C03642=1083.822,-32.819,444.005,174.181,18.899,153.143
C03643=1083.816,-33.092,444.020,174.180,18.898,153.143
C03644=1083.809,-33.364,444.033,174.179,18.896,153.143
C03645=1083.803,-33.637,444.048,174.176,18.894,153.143
C03646=1083.796,-33.887,444.060,174.175,18.892,153.143
C03647=1083.791,-34.136,444.072,174.174,18.890,153.143
C03648=1083.785,-34.386,444.084,174.172,18.888,153.143
C03649=1083.779,-34.636,444.097,174.171,18.886,153.143
C03650=1083.773,-34.885,444.109,174.170,18.885,153.143
C03651=1083.767,-35.135,444.122,174.168,18.882,153.143
C03652=1083.762,-35.384,444.134,174.166,18.881,153.143
C03653=1083.756,-35.634,444.147,174.165,18.879,153.143
C03654=1083.750,-35.884,444.159,174.163,18.877,153.142
C03655=1083.743,-36.133,444.172,174.162,18.876,153.142
C03656=1083.738,-36.382,444.184,174.161,18.874,153.142
C03657=1083.732,-36.632,444.197,174.159,18.872,153.142
C03658=1083.726,-36.882,444.209,174.157,18.870,153.142
C03659=1083.721,-37.131,444.221,174.156,18.868,153.142
C03660=1083.715,-37.381,444.234,174.154,18.866,153.142
C03661=1083.708,-37.631,444.246,174.153,18.865,153.142
C03662=1083.702,-37.881,444.259,174.152,18.863,153.142
C03663=1083.697,-38.130,444.271,174.150,18.861,153.142
C03664=1083.691,-38.380,444.283,174.149,18.859,153.142
C03665=1083.685,-38.630,444.296,174.147,18.857,153.142
C03666=1083.680,-38.879,444.308,174.145,18.856,153.142
C03667=1083.673,-39.128,444.320,174.144,18.854,153.141
C03668=1083.668,-39.378,444.333,174.143,18.852,153.141
C03669=1083.662,-39.628,444.345,174.141,18.851,153.141
C03670=1083.656,-39.877,444.357,174.140,18.849,153.141
C03671=1083.650,-40.127,444.369,174.139,18.847,153.141
C03672=1083.644,-40.377,444.381,174.137,18.845,153.141
C03673=1083.637,-40.627,444.393,174.135,18.844,153.141
C03674=1083.632,-40.876,444.405,174.134,18.842,153.141
C03675=1083.626,-41.126,444.418,174.132,18.840,153.141
C03676=1083.620,-41.376,444.430,174.131,18.838,153.141
C03677=1083.614,-41.625,444.442,174.130,18.837,153.141
C03678=1083.608,-41.875,444.454,174.128,18.835,153.141
C03679=1083.602,-42.124,444.466,174.127,18.833,153.141
C03680=1083.596,-42.374,444.479,174.125,18.831,153.141
C03681=1083.590,-42.623,444.491,174.123,18.830,153.141
C03682=1083.584,-42.874,444.502,174.122,18.828,153.140
C03683=1083.578,-43.123,444.515,174.121,18.826,153.140
C03684=1083.572,-43.372,444.527,174.119,18.825,153.140
C03685=1083.566,-43.622,444.539,174.118,18.823,153.140
C03686=1083.560,-43.872,444.552,174.117,18.821,153.140
C03687=1083.554,-44.121,444.563,174.115,18.819,153.140
C03688=1083.548,-44.371,444.576,174.113,18.817,153.140
C03689=1083.543,-44.621,444.588,174.111,18.816,153.140
C03690=1083.537,-44.870,444.599,174.110,18.814,153.140
C03691=1083.531,-45.120,444.612,174.109,18.812,153.140
C03692=1083.524,-45.370,444.624,174.107,18.811,153.140
C03693=1083.519,-45.619,444.636,174.106,18.809,153.140
C03694=1083.513,-45.869,444.648,174.105,18.807,153.140
C03695=1083.507,-46.119,444.660,174.103,18.806,153.139
C03696=1083.501,-46.368,444.672,174.102,18.804,153.139
C03697=1083.495,-46.618,444.684,174.099,18.802,153.139
C03698=1083.490,-46.867,444.695,174.098,18.801,153.139
C03699=1083.484,-47.117,444.708,174.097,18.799,153.139
C03700=1083.477,-47.367,444.720,174.095,18.797,153.139
C03701=1083.472,-47.616,444.732,174.094,18.795,153.139
C03702=1083.465,-47.866,444.743,174.093,18.794,153.139
C03703=1083.460,-48.116,444.756,174.091,18.792,153.139
C03704=1083.454,-48.365,444.768,174.090,18.790,153.139
C03705=1083.448,-48.615,444.780,174.088,18.789,153.139
C03706=1083.441,-48.888,444.793,174.086,18.787,153.139
C03707=1083.435,-49.160,444.806,174.085,18.785,153.139
C03708=1083.429,-49.433,444.819,174.084,18.783,153.139
C03709=1083.423,-49.706,444.832,174.081,18.781,153.139
C03710=1083.416,-49.956,444.844,174.080,18.779,153.139
C03711=1083.411,-50.206,444.855,174.079,18.778,153.139
C03712=1083.404,-50.455,444.867,174.077,18.776,153.138
C03713=1083.399,-50.705,444.880,174.076,18.775,153.138
C03714=1083.393,-50.955,444.891,174.074,18.773,153.138
C03715=1083.386,-51.204,444.903,174.073,18.771,153.138
C03716=1083.381,-51.453,444.915,174.071,18.770,153.138
C03717=1083.374,-51.704,444.926,174.070,18.768,153.138
C03718=1083.368,-51.953,444.938,174.069,18.766,153.138
C03719=1083.363,-52.203,444.950,174.067,18.764,153.138
C03720=1083.356,-52.453,444.962,174.065,18.763,153.138
C03721=1083.349,-52.702,444.974,174.064,18.761,153.138
C03722=1083.344,-52.952,444.985,174.062,18.760,153.138
C03723=1083.338,-53.202,444.997,174.061,18.758,153.138
C03724=1083.332,-53.451,445.008,174.059,18.757,153.138
C03725=1083.325,-53.701,445.020,174.058,18.755,153.138
C03726=1083.319,-53.951,445.032,174.057,18.754,153.138
C03727=1083.314,-54.200,445.043,174.055,18.752,153.138
C03728=1083.307,-54.450,445.055,174.054,18.751,153.138
C03729=1083.302,-54.699,445.067,174.052,18.749,153.138
C03730=1083.295,-54.949,445.079,174.051,18.747,153.138
C03731=1083.289,-55.199,445.090,174.049,18.746,153.138
C03732=1083.283,-55.448,445.101,174.047,18.744,153.138
C03733=1083.277,-55.699,445.113,174.046,18.742,153.138
C03734=1083.271,-55.947,445.125,174.044,18.740,153.138
C03735=1083.265,-56.198,445.136,174.043,18.739,153.137
C03736=1083.260,-56.447,445.148,174.042,18.737,153.137
C03737=1083.253,-56.697,445.160,174.040,18.736,153.137
C03738=1083.247,-56.947,445.172,174.039,18.734,153.137
C03739=1083.241,-57.196,445.182,174.037,18.733,153.137
C03740=1083.235,-57.446,445.195,174.036,18.731,153.137
C03741=1083.229,-57.695,445.206,174.034,18.730,153.137
C03742=1083.223,-57.945,445.218,174.033,18.728,153.137
C03743=1083.217,-58.194,445.229,174.032,18.726,153.137
C03744=1083.211,-58.444,445.241,174.030,18.725,153.137
C03745=1083.205,-58.694,445.252,174.029,18.723,153.137
C03746=1083.199,-58.944,445.263,174.026,18.721,153.137
C03747=1083.193,-59.193,445.275,174.025,18.720,153.137
C03748=1083.187,-59.443,445.286,174.024,18.718,153.137
C03749=1083.181,-59.692,445.298,174.022,18.717,153.137
C03750=1083.175,-59.942,445.310,174.021,18.715,153.137
C03751=1083.169,-60.192,445.320,174.019,18.714,153.137
C03752=1083.163,-60.441,445.332,174.018,18.712,153.137
C03753=1083.158,-60.691,445.344,174.016,18.711,153.137
C03754=1083.151,-60.941,445.356,174.015,18.709,153.137
C03755=1083.145,-61.190,445.367,174.013,18.708,153.137
C03756=1083.139,-61.441,445.378,174.012,18.706,153.137
C03757=1083.133,-61.689,445.390,174.011,18.704,153.137
C03758=1083.127,-61.940,445.401,174.009,18.703,153.137
C03759=1083.121,-62.189,445.412,174.008,18.701,153.137
C03760=1083.115,-62.439,445.424,174.006,18.700,153.137
C03761=1083.109,-62.688,445.435,174.005,18.698,153.137
C03762=1083.103,-62.939,445.446,174.003,18.697,153.137
C03763=1083.097,-63.188,445.459,174.002,18.695,153.137
C03764=1083.092,-63.437,445.469,174.001,18.694,153.137
C03765=1083.085,-63.688,445.481,173.998,18.692,153.137
C03766=1083.079,-63.936,445.492,173.997,18.690,153.137
C03767=1083.073,-64.187,445.504,173.995,18.689,153.137
C03768=1083.067,-64.436,445.514,173.994,18.687,153.136
C03769=1083.062,-64.687,445.526,173.993,18.686,153.136
C03770=1083.055,-64.960,445.538,173.991,18.684,153.136
C03771=1083.048,-65.235,445.551,173.990,18.682,153.136
C03772=1083.042,-65.508,445.563,173.988,18.681,153.136
C03773=1083.035,-65.782,445.576,173.986,18.679,153.136
C03774=1083.029,-66.032,445.587,173.985,18.677,153.136
C03775=1083.023,-66.282,445.598,173.983,18.676,153.136
C03776=1083.018,-66.531,445.610,173.982,18.674,153.136
C03777=1083.011,-66.782,445.621,173.980,18.673,153.136
C03778=1083.006,-67.031,445.632,173.979,18.671,153.136
C03779=1083.000,-67.280,445.643,173.977,18.670,153.136
C03780=1082.994,-67.531,445.654,173.976,18.668,153.136
C03781=1082.988,-67.780,445.665,173.974,18.667,153.136
C03782=1082.982,-68.029,445.677,173.973,18.666,153.136
C03783=1082.975,-68.279,445.688,173.971,18.664,153.136
C03784=1082.970,-68.529,445.700,173.970,18.663,153.136
C03785=1082.965,-68.779,445.710,173.968,18.661,153.136
C03786=1082.958,-69.029,445.722,173.967,18.659,153.136
C03787=1082.953,-69.278,445.733,173.966,18.658,153.136
C03788=1082.947,-69.527,445.744,173.964,18.656,153.136
C03789=1082.940,-69.777,445.755,173.963,18.655,153.136
C03790=1082.935,-70.027,445.766,173.961,18.653,153.136
C03791=1082.929,-70.276,445.777,173.960,18.652,153.136
C03792=1082.922,-70.526,445.788,173.958,18.650,153.136
C03793=1082.917,-70.776,445.800,173.957,18.649,153.136
C03794=1082.912,-71.026,445.811,173.955,18.648,153.136
C03795=1082.905,-71.276,445.822,173.954,18.646,153.136
C03796=1082.900,-71.525,445.833,173.952,18.645,153.136
C03797=1082.894,-71.774,445.845,173.951,18.643,153.136
C03798=1082.887,-72.024,445.856,173.950,18.642,153.136
C03799=1082.881,-72.274,445.867,173.948,18.640,153.136
C03800=1082.876,-72.523,445.878,173.947,18.638,153.136
C03801=1082.869,-72.774,445.889,173.945,18.637,153.136
C03802=1082.864,-73.023,445.900,173.944,18.636,153.136
C03803=1082.858,-73.273,445.911,173.942,18.634,153.136
C03804=1082.852,-73.522,445.921,173.941,18.633,153.136
C03805=1082.846,-73.772,445.933,173.939,18.631,153.136
C03806=1082.840,-74.022,445.944,173.938,18.630,153.136
C03807=1082.834,-74.271,445.954,173.936,18.628,153.136
C03808=1082.828,-74.521,445.966,173.935,18.627,153.136
C03809=1082.822,-74.771,445.977,173.933,18.626,153.136
C03810=1082.817,-75.020,445.987,173.932,18.624,153.136
C03811=1082.810,-75.271,445.999,173.930,18.623,153.136
C03812=1082.804,-75.520,446.010,173.929,18.622,153.136
C03813=1082.799,-75.770,446.020,173.927,18.620,153.136
C03814=1082.793,-76.019,446.031,173.926,18.619,153.136
C03815=1082.786,-76.269,446.042,173.924,18.617,153.136
C03816=1082.780,-76.518,446.053,173.923,18.616,153.136
C03817=1082.774,-76.768,446.064,173.921,18.614,153.136
C03818=1082.768,-77.018,446.075,173.920,18.613,153.136
C03819=1082.762,-77.268,446.086,173.918,18.611,153.136
C03820=1082.757,-77.518,446.096,173.917,18.610,153.136
C03821=1082.751,-77.768,446.107,173.915,18.609,153.136
C03822=1082.744,-78.017,446.117,173.914,18.607,153.136
C03823=1082.738,-78.267,446.128,173.913,18.606,153.136
C03824=1082.733,-78.516,446.139,173.911,18.605,153.136
C03825=1082.726,-78.766,446.150,173.909,18.603,153.136
C03826=1082.721,-79.016,446.161,173.908,18.602,153.136
C03827=1082.715,-79.265,446.172,173.906,18.601,153.136
C03828=1082.708,-79.514,446.183,173.905,18.599,153.136
C03829=1082.702,-79.765,446.194,173.903,18.598,153.136
C03830=1082.697,-80.015,446.204,173.902,18.597,153.136
C03831=1082.691,-80.264,446.215,173.900,18.595,153.136
C03832=1082.684,-80.513,446.225,173.899,18.594,153.136
C03833=1082.678,-80.764,446.236,173.897,18.592,153.136
C03834=1082.671,-81.040,446.248,173.896,18.591,153.136
C03835=1082.665,-81.317,446.260,173.894,18.589,153.136
C03836=1082.658,-81.593,446.271,173.893,18.588,153.136
C03837=1082.651,-81.869,446.283,173.891,18.587,153.136
C03838=1082.645,-82.119,446.294,173.890,18.586,153.136
C03839=1082.638,-82.368,446.305,173.888,18.584,153.136
C03840=1082.633,-82.618,446.315,173.887,18.583,153.136
C03841=1082.627,-82.867,446.326,173.885,18.582,153.136
C03842=1082.621,-83.117,446.336,173.884,18.580,153.136
C03843=1082.614,-83.367,446.347,173.882,18.579,153.136
C03844=1082.609,-83.617,446.358,173.880,18.578,153.136
C03845=1082.602,-83.866,446.368,173.879,18.577,153.136
C03846=1082.596,-84.116,446.379,173.877,18.575,153.136
C03847=1082.590,-84.366,446.390,173.876,18.574,153.136
C03848=1082.584,-84.616,446.400,173.874,18.573,153.136
C03849=1082.578,-84.865,446.411,173.873,18.571,153.136
C03850=1082.572,-85.114,446.421,173.871,18.570,153.136
C03851=1082.566,-85.365,446.432,173.870,18.568,153.136
C03852=1082.560,-85.615,446.443,173.868,18.567,153.137
C03853=1082.553,-85.864,446.453,173.867,18.566,153.137
C03854=1082.548,-86.114,446.463,173.865,18.565,153.137
C03855=1082.541,-86.364,446.474,173.863,18.563,153.137
C03856=1082.535,-86.613,446.484,173.862,18.562,153.137
C03857=1082.530,-86.863,446.495,173.861,18.561,153.137
C03858=1082.523,-87.112,446.505,173.859,18.560,153.137
C03859=1082.518,-87.362,446.516,173.858,18.559,153.137
C03860=1082.511,-87.612,446.526,173.856,18.558,153.137
C03861=1082.505,-87.862,446.537,173.855,18.556,153.137
C03862=1082.499,-88.111,446.547,173.853,18.555,153.137
C03863=1082.493,-88.361,446.557,173.852,18.554,153.137
C03864=1082.487,-88.611,446.568,173.850,18.553,153.137
C03865=1082.481,-88.860,446.578,173.849,18.551,153.137
C03866=1082.475,-89.111,446.589,173.847,18.550,153.137
C03867=1082.469,-89.360,446.600,173.846,18.549,153.137
C03868=1082.463,-89.609,446.610,173.844,18.548,153.137
C03869=1082.457,-89.860,446.620,173.842,18.546,153.137
C03870=1082.451,-90.109,446.630,173.841,18.545,153.137
C03871=1082.445,-90.359,446.641,173.840,18.544,153.137
C03872=1082.438,-90.609,446.651,173.838,18.543,153.137
C03873=1082.432,-90.858,446.662,173.837,18.541,153.137
C03874=1082.426,-91.108,446.672,173.835,18.540,153.137
C03875=1082.421,-91.357,446.682,173.834,18.539,153.137
C03876=1082.415,-91.608,446.693,173.832,18.538,153.137
C03877=1082.409,-91.857,446.703,173.831,18.536,153.137
C03878=1082.403,-92.107,446.713,173.829,18.535,153.138
C03879=1082.397,-92.356,446.723,173.827,18.534,153.138
C03880=1082.391,-92.607,446.734,173.826,18.533,153.138
C03881=1082.384,-92.856,446.744,173.824,18.532,153.138
C03882=1082.379,-93.106,446.754,173.823,18.530,153.138
C03883=1082.372,-93.355,446.765,173.822,18.530,153.138
C03884=1082.367,-93.605,446.776,173.821,18.528,153.138
C03885=1082.360,-93.855,446.785,173.819,18.527,153.138
C03886=1082.355,-94.104,446.796,173.817,18.526,153.138
C03887=1082.349,-94.354,446.806,173.816,18.525,153.138
C03888=1082.343,-94.604,446.816,173.814,18.524,153.138
C03889=1082.337,-94.853,446.826,173.813,18.522,153.138
C03890=1082.331,-95.103,446.836,173.811,18.521,153.138
C03891=1082.325,-95.352,446.846,173.809,18.520,153.138
C03892=1082.319,-95.603,446.857,173.808,18.518,153.138
C03893=1082.312,-95.852,446.867,173.806,18.517,153.138
C03894=1082.307,-96.103,446.877,173.806,18.516,153.138
C03895=1082.300,-96.352,446.888,173.804,18.515,153.138
C03896=1082.295,-96.602,446.898,173.802,18.514,153.138
C03897=1082.288,-96.851,446.908,173.801,18.513,153.138
C03898=1082.282,-97.130,446.919,173.799,18.512,153.139
C03899=1082.275,-97.409,446.931,173.798,18.510,153.139
C03900=1082.269,-97.687,446.942,173.796,18.509,153.139
C03901=1082.262,-97.966,446.953,173.794,18.508,153.139
C03902=1082.256,-98.216,446.963,173.793,18.507,153.139
C03903=1082.250,-98.465,446.974,173.791,18.506,153.139
C03904=1082.244,-98.715,446.983,173.790,18.505,153.139
C03905=1082.238,-98.965,446.993,173.788,18.504,153.139
C03906=1082.232,-99.214,447.004,173.786,18.502,153.139
C03907=1082.225,-99.464,447.013,173.785,18.501,153.139
C03908=1082.219,-99.714,447.023,173.783,18.500,153.139
C03909=1082.214,-99.963,447.034,173.781,18.499,153.139
C03910=1082.207,-100.213,447.043,173.781,18.498,153.139
C03911=1082.201,-100.462,447.054,173.779,18.497,153.139
C03912=1082.195,-100.713,447.064,173.777,18.496,153.140
C03913=1082.189,-100.963,447.074,173.776,18.495,153.140
C03914=1082.182,-101.213,447.083,173.774,18.494,153.140
C03915=1082.177,-101.462,447.094,173.773,18.493,153.140
C03916=1082.171,-101.712,447.104,173.771,18.492,153.140
C03917=1082.164,-101.962,447.113,173.769,18.491,153.140
C03918=1082.158,-102.211,447.123,173.768,18.490,153.140
C03919=1082.152,-102.461,447.134,173.767,18.489,153.140
C03920=1082.146,-102.711,447.143,173.765,18.487,153.140
C03921=1082.140,-102.960,447.153,173.764,18.486,153.140
C03922=1082.134,-103.210,447.163,173.762,18.485,153.140
C03923=1082.128,-103.460,447.173,173.760,18.484,153.140
C03924=1082.122,-103.710,447.183,173.759,18.483,153.141
C03925=1082.116,-103.959,447.193,173.758,18.482,153.141
C03926=1082.109,-104.209,447.203,173.756,18.481,153.141
C03927=1082.104,-104.459,447.213,173.755,18.480,153.141
C03928=1082.098,-104.709,447.222,173.753,18.479,153.141
C03929=1082.091,-104.958,447.233,173.751,18.478,153.141
C03930=1082.085,-105.208,447.242,173.750,18.477,153.141
C03931=1082.080,-105.458,447.252,173.748,18.476,153.141
C03932=1082.074,-105.707,447.262,173.747,18.475,153.141
C03933=1082.067,-105.957,447.271,173.746,18.474,153.141
C03934=1082.061,-106.206,447.282,173.744,18.473,153.141
C03935=1082.055,-106.456,447.291,173.742,18.472,153.141
C03936=1082.049,-106.706,447.302,173.741,18.471,153.142
C03937=1082.043,-106.956,447.311,173.739,18.470,153.142
C03938=1082.037,-107.206,447.321,173.738,18.470,153.142
C03939=1082.031,-107.456,447.330,173.736,18.469,153.142
C03940=1082.024,-107.705,447.340,173.735,18.467,153.142
C03941=1082.018,-107.955,447.350,173.733,18.466,153.142
C03942=1082.013,-108.205,447.360,173.732,18.465,153.142
C03943=1082.007,-108.455,447.370,173.730,18.464,153.142
C03944=1082.000,-108.704,447.379,173.729,18.464,153.142
C03945=1081.994,-108.954,447.389,173.727,18.463,153.142
C03946=1081.988,-109.204,447.398,173.726,18.462,153.142
C03947=1081.982,-109.453,447.409,173.724,18.461,153.143
C03948=1081.975,-109.703,447.418,173.722,18.460,153.143
C03949=1081.970,-109.952,447.428,173.721,18.459,153.143
C03950=1081.964,-110.202,447.437,173.720,18.458,153.143
C03951=1081.957,-110.452,447.447,173.718,18.457,153.143
C03952=1081.951,-110.701,447.456,173.716,18.456,153.143
C03953=1081.945,-110.951,447.466,173.715,18.455,153.143
C03954=1081.940,-111.201,447.476,173.713,18.454,153.143
C03955=1081.934,-111.451,447.486,173.712,18.453,153.143
C03956=1081.927,-111.701,447.495,173.711,18.452,153.144
C03957=1081.921,-111.951,447.505,173.709,18.451,153.144
C03958=1081.915,-112.201,447.514,173.707,18.450,153.144
C03959=1081.909,-112.450,447.524,173.705,18.449,153.144
C03960=1081.903,-112.700,447.533,173.704,18.448,153.144
C03961=1081.896,-112.950,447.543,173.703,18.448,153.144
C03962=1081.889,-113.225,447.553,173.701,18.447,153.144
C03963=1081.883,-113.500,447.564,173.700,18.446,153.144
C03964=1081.877,-113.775,447.575,173.698,18.445,153.145
C03965=1081.870,-114.051,447.585,173.696,18.444,153.145
C03966=1081.864,-114.300,447.595,173.694,18.443,153.145
C03967=1081.857,-114.550,447.605,173.693,18.442,153.145
C03968=1081.851,-114.800,447.614,173.691,18.441,153.145
C03969=1081.846,-115.049,447.623,173.689,18.440,153.145
C03970=1081.839,-115.299,447.633,173.688,18.440,153.145
C03971=1081.833,-115.549,447.642,173.687,18.439,153.145
C03972=1081.827,-115.798,447.652,173.685,18.438,153.145
C03973=1081.821,-116.048,447.662,173.683,18.437,153.146
C03974=1081.815,-116.298,447.671,173.681,18.436,153.146
C03975=1081.808,-116.548,447.680,173.681,18.436,153.146
C03976=1081.802,-116.797,447.690,173.679,18.435,153.146
C03977=1081.796,-117.047,447.699,173.677,18.434,153.146
C03978=1081.789,-117.297,447.709,173.675,18.433,153.146
C03979=1081.784,-117.546,447.718,173.675,18.432,153.146
C03980=1081.778,-117.796,447.727,173.673,18.431,153.146
C03981=1081.772,-118.046,447.736,173.671,18.431,153.147
C03982=1081.766,-118.296,447.746,173.669,18.430,153.147
C03983=1081.759,-118.546,447.756,173.668,18.429,153.147
C03984=1081.753,-118.796,447.765,173.667,18.428,153.147
C03985=1081.747,-119.045,447.775,173.665,18.427,153.147
C03986=1081.741,-119.295,447.784,173.663,18.426,153.147
C03987=1081.735,-119.544,447.793,173.661,18.426,153.148
C03988=1081.729,-119.794,447.802,173.661,18.425,153.148
C03989=1081.723,-120.044,447.811,173.659,18.424,153.148
C03990=1081.716,-120.294,447.821,173.657,18.423,153.148
C03991=1081.710,-120.544,447.830,173.655,18.423,153.148
C03992=1081.704,-120.794,447.840,173.654,18.422,153.148
C03993=1081.698,-121.043,447.849,173.653,18.421,153.148
C03994=1081.692,-121.293,447.859,173.651,18.420,153.148
C03995=1081.686,-121.543,447.867,173.649,18.420,153.149
C03996=1081.679,-121.792,447.877,173.648,18.419,153.149
C03997=1081.673,-122.042,447.886,173.647,18.418,153.149
C03998=1081.667,-122.292,447.896,173.645,18.417,153.149
C03999=1081.662,-122.541,447.905,173.643,18.417,153.149
C04000=1081.656,-122.792,447.914,173.641,18.416,153.149
C04001=1081.649,-123.041,447.923,173.641,18.415,153.149
C04002=1081.643,-123.291,447.932,173.639,18.414,153.149
C04003=1081.636,-123.541,447.942,173.637,18.414,153.150
C04004=1081.631,-123.791,447.951,173.635,18.413,153.150
C04005=1081.625,-124.040,447.960,173.634,18.412,153.150
C04006=1081.618,-124.290,447.969,173.632,18.412,153.150
C04007=1081.612,-124.539,447.978,173.631,18.411,153.150
C04008=1081.606,-124.790,447.987,173.629,18.410,153.150
C04009=1081.600,-125.040,447.997,173.628,18.410,153.151
C04010=1081.594,-125.288,448.006,173.626,18.409,153.151
C04011=1081.587,-125.538,448.015,173.625,18.408,153.151
C04012=1081.582,-125.789,448.024,173.623,18.407,153.151
C04013=1081.575,-126.038,448.033,173.622,18.407,153.151
C04014=1081.568,-126.288,448.042,173.620,18.406,153.151
C04015=1081.563,-126.538,448.051,173.618,18.405,153.152
C04016=1081.557,-126.787,448.061,173.616,18.404,153.152
C04017=1081.551,-127.037,448.070,173.615,18.404,153.152
C04018=1081.544,-127.287,448.079,173.614,18.403,153.152
C04019=1081.538,-127.537,448.088,173.612,18.402,153.152
C04020=1081.532,-127.787,448.097,173.610,18.402,153.152
C04021=1081.527,-128.037,448.106,173.609,18.401,153.152
C04022=1081.523,-128.292,448.116,173.608,18.400,153.152
C04023=1081.523,-128.548,448.128,173.607,18.397,153.152
C04024=1081.527,-128.801,448.141,173.607,18.393,153.152
C04025=1081.534,-129.053,448.155,173.607,18.389,153.151
C04026=1081.134,-129.075,448.015,173.562,18.508,153.181
C04027=1081.127,-128.823,448.002,173.562,18.512,153.182
C04028=1081.123,-128.569,447.989,173.563,18.516,153.182
C04029=1081.123,-128.314,447.977,173.563,18.519,153.183
C04030=1081.126,-128.059,447.967,173.565,18.521,153.183
C04031=1081.132,-127.809,447.957,173.566,18.522,153.183
C04032=1081.138,-127.559,447.949,173.568,18.522,153.183
C04033=1081.144,-127.309,447.939,173.569,18.523,153.182
C04034=1081.150,-127.059,447.929,173.571,18.524,153.182
C04035=1081.156,-126.810,447.922,173.573,18.524,153.182
C04036=1081.162,-126.560,447.912,173.575,18.525,153.182
C04037=1081.169,-126.310,447.902,173.575,18.526,153.182
C04038=1081.175,-126.061,447.893,173.577,18.526,153.182
C04039=1081.181,-125.810,447.885,173.579,18.527,153.182
C04040=1081.187,-125.561,447.875,173.581,18.528,153.181
C04041=1081.193,-125.311,447.866,173.582,18.528,153.181
C04042=1081.200,-125.061,447.858,173.584,18.529,153.181
C04043=1081.206,-124.811,447.848,173.585,18.530,153.181
C04044=1081.212,-124.562,447.838,173.587,18.531,153.181
C04045=1081.218,-124.312,447.829,173.588,18.531,153.181
C04046=1081.224,-124.062,447.821,173.590,18.532,153.180
C04047=1081.230,-123.813,447.811,173.592,18.533,153.180
C04048=1081.236,-123.563,447.802,173.593,18.534,153.180
C04049=1081.243,-123.313,447.792,173.594,18.534,153.180
C04050=1081.249,-123.063,447.783,173.596,18.535,153.180
C04051=1081.255,-122.814,447.775,173.598,18.536,153.180
C04052=1081.261,-122.564,447.765,173.599,18.537,153.180
C04053=1081.267,-122.314,447.756,173.600,18.537,153.179
C04054=1081.273,-122.064,447.746,173.602,18.538,153.179
C04055=1081.279,-121.814,447.737,173.604,18.539,153.179
C04056=1081.285,-121.564,447.728,173.606,18.540,153.179
C04057=1081.291,-121.315,447.718,173.607,18.541,153.179
C04058=1081.298,-121.066,447.710,173.608,18.541,153.179
C04059=1081.304,-120.816,447.700,173.610,18.542,153.179
C04060=1081.310,-120.566,447.690,173.612,18.543,153.178
C04061=1081.316,-120.316,447.682,173.613,18.544,153.178
C04062=1081.322,-120.066,447.672,173.614,18.544,153.178
C04063=1081.328,-119.817,447.663,173.616,18.545,153.178
C04064=1081.334,-119.567,447.653,173.618,18.546,153.178
C04065=1081.341,-119.317,447.644,173.620,18.547,153.178
C04066=1081.347,-119.068,447.635,173.621,18.548,153.178
C04067=1081.353,-118.818,447.625,173.622,18.548,153.178
C04068=1081.359,-118.567,447.616,173.624,18.549,153.177
C04069=1081.365,-118.318,447.607,173.626,18.550,153.177
C04070=1081.371,-118.068,447.597,173.627,18.551,153.177
C04071=1081.377,-117.819,447.588,173.629,18.552,153.177
C04072=1081.383,-117.569,447.578,173.630,18.552,153.177
C04073=1081.389,-117.319,447.569,173.632,18.553,153.177
C04074=1081.396,-117.069,447.559,173.633,18.554,153.177
C04075=1081.402,-116.819,447.550,173.635,18.555,153.177
C04076=1081.408,-116.570,447.540,173.636,18.556,153.176
C04077=1081.414,-116.320,447.530,173.638,18.557,153.176
C04078=1081.421,-116.070,447.522,173.639,18.558,153.176
C04079=1081.427,-115.821,447.512,173.641,18.559,153.176
C04080=1081.433,-115.571,447.503,173.643,18.559,153.176
C04081=1081.439,-115.322,447.493,173.644,18.560,153.176
C04082=1081.445,-115.071,447.484,173.645,18.561,153.176
C04083=1081.451,-114.821,447.475,173.647,18.562,153.176
C04084=1081.457,-114.572,447.465,173.649,18.563,153.175
C04085=1081.463,-114.322,447.456,173.651,18.564,153.175
C04086=1081.469,-114.072,447.446,173.652,18.565,153.175
C04087=1081.476,-113.796,447.435,173.654,18.566,153.175
C04088=1081.483,-113.521,447.424,173.656,18.567,153.175
C04089=1081.490,-113.246,447.414,173.657,18.568,153.175
C04090=1081.497,-112.971,447.403,173.659,18.569,153.175
C04091=1081.503,-112.721,447.394,173.660,18.569,153.175
C04092=1081.509,-112.472,447.384,173.661,18.570,153.175
C04093=1081.514,-112.222,447.374,173.663,18.571,153.174
C04094=1081.520,-111.972,447.365,173.665,18.572,153.174
C04095=1081.526,-111.722,447.355,173.667,18.573,153.174
C04096=1081.532,-111.472,447.346,173.667,18.574,153.174
C04097=1081.539,-111.223,447.336,173.669,18.575,153.174
C04098=1081.545,-110.973,447.326,173.671,18.576,153.174
C04099=1081.551,-110.723,447.317,173.672,18.577,153.174
C04100=1081.557,-110.473,447.307,173.674,18.578,153.174
C04101=1081.563,-110.223,447.298,173.676,18.579,153.174
C04102=1081.570,-109.974,447.288,173.677,18.579,153.173
C04103=1081.576,-109.724,447.279,173.678,18.580,153.173
C04104=1081.582,-109.475,447.268,173.680,18.581,153.173
C04105=1081.588,-109.225,447.259,173.682,18.582,153.173
C04106=1081.595,-108.975,447.249,173.683,18.583,153.173
C04107=1081.600,-108.725,447.239,173.685,18.584,153.173
C04108=1081.606,-108.475,447.229,173.686,18.585,153.173
C04109=1081.612,-108.225,447.220,173.687,18.586,153.173
C04110=1081.618,-107.975,447.210,173.689,18.587,153.173
C04111=1081.625,-107.726,447.201,173.691,18.588,153.173
C04112=1081.631,-107.476,447.190,173.692,18.589,153.173
C04113=1081.637,-107.227,447.181,173.694,18.590,153.172
C04114=1081.643,-106.977,447.171,173.695,18.591,153.172
C04115=1081.649,-106.727,447.161,173.697,18.592,153.172
C04116=1081.655,-106.477,447.152,173.698,18.593,153.172
C04117=1081.661,-106.227,447.142,173.700,18.594,153.172
C04118=1081.668,-105.978,447.132,173.701,18.595,153.172
C04119=1081.674,-105.728,447.122,173.703,18.596,153.172
C04120=1081.679,-105.478,447.112,173.705,18.597,153.172
C04121=1081.685,-105.229,447.103,173.706,18.598,153.172
C04122=1081.691,-104.980,447.093,173.707,18.599,153.172
C04123=1081.698,-104.730,447.083,173.709,18.600,153.172
C04124=1081.703,-104.480,447.073,173.711,18.601,153.172
C04125=1081.709,-104.230,447.063,173.712,18.602,153.171
C04126=1081.715,-103.980,447.054,173.714,18.603,153.171
C04127=1081.722,-103.731,447.043,173.716,18.604,153.171
C04128=1081.728,-103.480,447.033,173.716,18.605,153.171
C04129=1081.734,-103.231,447.023,173.718,18.606,153.171
C04130=1081.740,-102.981,447.013,173.720,18.607,153.171
C04131=1081.747,-102.732,447.003,173.721,18.608,153.171
C04132=1081.752,-102.481,446.993,173.723,18.609,153.171
C04133=1081.758,-102.232,446.984,173.724,18.611,153.171
C04134=1081.765,-101.982,446.973,173.726,18.612,153.171
C04135=1081.771,-101.733,446.964,173.727,18.613,153.171
C04136=1081.776,-101.483,446.954,173.729,18.614,153.171
C04137=1081.783,-101.233,446.943,173.730,18.615,153.171
C04138=1081.789,-100.984,446.934,173.732,18.616,153.170
C04139=1081.794,-100.733,446.924,173.733,18.617,153.170
C04140=1081.801,-100.484,446.913,173.735,18.618,153.170
C04141=1081.807,-100.235,446.904,173.737,18.620,153.170
C04142=1081.812,-99.984,446.894,173.738,18.621,153.170
C04143=1081.819,-99.735,446.883,173.739,18.621,153.170
C04144=1081.825,-99.485,446.874,173.741,18.622,153.170
C04145=1081.831,-99.236,446.864,173.742,18.624,153.170
C04146=1081.837,-98.986,446.853,173.744,18.625,153.170
C04147=1081.843,-98.736,446.844,173.746,18.626,153.170
C04148=1081.850,-98.486,446.834,173.747,18.627,153.170
C04149=1081.856,-98.236,446.823,173.749,18.628,153.170
C04150=1081.862,-97.987,446.813,173.750,18.629,153.170
C04151=1081.868,-97.709,446.802,173.752,18.630,153.169
C04152=1081.876,-97.430,446.791,173.753,18.632,153.169
C04153=1081.882,-97.151,446.780,173.755,18.633,153.169
C04154=1081.889,-96.872,446.768,173.757,18.634,153.169
C04155=1081.894,-96.622,446.758,173.758,18.635,153.169
C04156=1081.901,-96.372,446.748,173.760,18.637,153.169
C04157=1081.906,-96.123,446.737,173.761,18.638,153.169
C04158=1081.912,-95.873,446.728,173.763,18.639,153.169
C04159=1081.918,-95.623,446.717,173.765,18.640,153.169
C04160=1081.924,-95.374,446.707,173.765,18.641,153.169
C04161=1081.930,-95.124,446.697,173.767,18.642,153.169
C04162=1081.936,-94.875,446.687,173.769,18.643,153.169
C04163=1081.942,-94.624,446.676,173.770,18.645,153.169
C04164=1081.949,-94.375,446.666,173.772,18.646,153.169
C04165=1081.954,-94.125,446.656,173.773,18.647,153.169
C04166=1081.961,-93.875,446.645,173.775,18.649,153.169
C04167=1081.966,-93.625,446.635,173.776,18.650,153.169
C04168=1081.973,-93.376,446.625,173.778,18.651,153.169
C04169=1081.978,-93.126,446.615,173.780,18.652,153.169
C04170=1081.985,-92.877,446.604,173.781,18.654,153.169
C04171=1081.990,-92.627,446.594,173.783,18.655,153.168
C04172=1081.996,-92.377,446.584,173.783,18.656,153.169
C04173=1082.003,-92.127,446.574,173.785,18.657,153.168
C04174=1082.009,-91.877,446.563,173.786,18.658,153.168
C04175=1082.015,-91.628,446.552,173.788,18.659,153.168
C04176=1082.020,-91.378,446.542,173.790,18.661,153.168
C04177=1082.027,-91.129,446.532,173.791,18.662,153.168
C04178=1082.032,-90.879,446.522,173.793,18.663,153.168
C04179=1082.039,-90.629,446.511,173.794,18.664,153.168
C04180=1082.044,-90.379,446.501,173.796,18.666,153.168
C04181=1082.051,-90.129,446.491,173.797,18.667,153.168
C04182=1082.057,-89.880,446.480,173.799,18.668,153.168
C04183=1082.063,-89.630,446.470,173.801,18.669,153.168
C04184=1082.069,-89.381,446.459,173.802,18.671,153.168
C04185=1082.074,-89.131,446.448,173.803,18.671,153.168
C04186=1082.081,-88.881,446.439,173.804,18.673,153.168
C04187=1082.087,-88.631,446.428,173.806,18.674,153.168
C04188=1082.093,-88.381,446.418,173.807,18.675,153.168
C04189=1082.099,-88.132,446.407,173.809,18.676,153.168
C04190=1082.105,-87.883,446.397,173.811,18.678,153.168
C04191=1082.111,-87.633,446.387,173.812,18.679,153.168
C04192=1082.117,-87.383,446.376,173.814,18.681,153.168
C04193=1082.124,-87.133,446.365,173.815,18.682,153.168
C04194=1082.129,-86.883,446.355,173.817,18.683,153.168
C04195=1082.136,-86.634,446.345,173.818,18.685,153.168
C04196=1082.141,-86.384,446.334,173.820,18.686,153.168
C04197=1082.148,-86.134,446.323,173.821,18.687,153.168
C04198=1082.154,-85.884,446.313,173.823,18.688,153.168
C04199=1082.160,-85.635,446.302,173.824,18.690,153.168
C04200=1082.166,-85.386,446.292,173.826,18.691,153.167
C04201=1082.171,-85.136,446.282,173.828,18.692,153.167
C04202=1082.178,-84.886,446.271,173.828,18.693,153.168
C04203=1082.184,-84.636,446.260,173.830,18.694,153.167
C04204=1082.190,-84.387,446.249,173.831,18.696,153.167
C04205=1082.195,-84.137,446.239,173.833,18.697,153.167
C04206=1082.202,-83.887,446.229,173.834,18.698,153.167
C04207=1082.208,-83.637,446.218,173.836,18.699,153.167
C04208=1082.215,-83.388,446.207,173.838,18.701,153.167
C04209=1082.220,-83.138,446.197,173.839,18.702,153.167
C04210=1082.226,-82.888,446.186,173.841,18.703,153.167
C04211=1082.233,-82.639,446.176,173.842,18.705,153.167
C04212=1082.239,-82.389,446.165,173.844,18.706,153.167
C04213=1082.244,-82.140,446.154,173.845,18.707,153.167
C04214=1082.251,-81.889,446.144,173.847,18.709,153.167
C04215=1082.258,-81.613,446.131,173.848,18.710,153.167
C04216=1082.265,-81.337,446.120,173.850,18.712,153.167
C04217=1082.271,-81.061,446.108,173.851,18.713,153.167
C04218=1082.278,-80.784,446.096,173.854,18.715,153.167
C04219=1082.285,-80.534,446.085,173.855,18.716,153.167
C04220=1082.290,-80.284,446.075,173.857,18.718,153.167
C04221=1082.296,-80.035,446.064,173.858,18.719,153.167
C04222=1082.303,-79.785,446.054,173.860,18.720,153.167
C04223=1082.309,-79.535,446.043,173.861,18.722,153.167
C04224=1082.314,-79.286,446.032,173.862,18.723,153.167
C04225=1082.320,-79.036,446.021,173.864,18.724,153.167
C04226=1082.326,-78.786,446.010,173.865,18.725,153.167
C04227=1082.332,-78.537,445.999,173.866,18.727,153.167
C04228=1082.338,-78.287,445.989,173.868,18.728,153.167
C04229=1082.345,-78.037,445.978,173.870,18.729,153.167
C04230=1082.350,-77.787,445.967,173.871,18.731,153.167
C04231=1082.356,-77.538,445.956,173.872,18.732,153.167
C04232=1082.362,-77.288,445.945,173.874,18.734,153.167
C04233=1082.368,-77.038,445.934,173.876,18.735,153.167
C04234=1082.374,-76.788,445.923,173.877,18.736,153.167
C04235=1082.380,-76.539,445.913,173.878,18.738,153.167
C04236=1082.387,-76.289,445.902,173.880,18.740,153.167
C04237=1082.393,-76.040,445.891,173.881,18.741,153.167
C04238=1082.398,-75.790,445.880,173.883,18.742,153.167
C04239=1082.404,-75.541,445.869,173.884,18.744,153.167
C04240=1082.410,-75.290,445.858,173.886,18.745,153.167
C04241=1082.416,-75.041,445.847,173.887,18.747,153.167
C04242=1082.422,-74.791,445.836,173.889,18.748,153.167
C04243=1082.429,-74.542,445.826,173.890,18.749,153.167
C04244=1082.435,-74.292,445.815,173.892,18.751,153.167
C04245=1082.440,-74.043,445.804,173.893,18.752,153.167
C04246=1082.447,-73.792,445.793,173.895,18.754,153.167
C04247=1082.453,-73.543,445.782,173.896,18.755,153.167
C04248=1082.458,-73.293,445.771,173.898,18.757,153.167
C04249=1082.465,-73.043,445.760,173.899,18.758,153.167
C04250=1082.470,-72.793,445.748,173.901,18.759,153.167
C04251=1082.475,-72.544,445.737,173.902,18.761,153.167
C04252=1082.481,-72.294,445.726,173.904,18.762,153.167
C04253=1082.487,-72.044,445.715,173.905,18.764,153.167
C04254=1082.493,-71.795,445.704,173.906,18.766,153.167
C04255=1082.499,-71.545,445.693,173.908,18.767,153.167
C04256=1082.505,-71.295,445.682,173.909,18.769,153.167
C04257=1082.511,-71.046,445.671,173.911,18.770,153.167
C04258=1082.517,-70.797,445.660,173.912,18.772,153.167
C04259=1082.523,-70.546,445.648,173.914,18.773,153.167
C04260=1082.529,-70.297,445.637,173.915,18.775,153.167
C04261=1082.535,-70.048,445.627,173.917,18.776,153.167
C04262=1082.540,-69.797,445.615,173.919,18.778,153.167
C04263=1082.546,-69.548,445.604,173.920,18.780,153.167
C04264=1082.552,-69.298,445.593,173.922,18.781,153.167
C04265=1082.558,-69.048,445.582,173.923,18.783,153.167
C04266=1082.564,-68.799,445.570,173.925,18.784,153.167
C04267=1082.570,-68.549,445.559,173.926,18.785,153.167
C04268=1082.576,-68.299,445.548,173.928,18.787,153.167
C04269=1082.582,-68.050,445.537,173.929,18.788,153.167
C04270=1082.587,-67.800,445.526,173.931,18.790,153.167
C04271=1082.593,-67.550,445.514,173.932,18.792,153.168
C04272=1082.600,-67.301,445.503,173.934,18.793,153.168
C04273=1082.606,-67.051,445.492,173.935,18.795,153.168
C04274=1082.612,-66.801,445.481,173.936,18.796,153.168
C04275=1082.617,-66.552,445.470,173.938,18.798,153.168
C04276=1082.624,-66.302,445.458,173.939,18.799,153.168
C04277=1082.629,-66.052,445.446,173.941,18.801,153.168
C04278=1082.635,-65.803,445.436,173.942,18.802,153.168
C04279=1082.642,-65.529,445.423,173.944,18.804,153.168
C04280=1082.649,-65.254,445.410,173.945,18.805,153.168
C04281=1082.655,-64.979,445.399,173.947,18.808,153.168
C04282=1082.661,-64.706,445.386,173.948,18.809,153.168
C04283=1082.667,-64.455,445.374,173.950,18.811,153.168
C04284=1082.673,-64.206,445.363,173.951,18.812,153.168
C04285=1082.679,-63.956,445.352,173.953,18.814,153.168
C04286=1082.685,-63.707,445.341,173.954,18.815,153.168
C04287=1082.691,-63.458,445.329,173.956,18.817,153.168
C04288=1082.698,-63.208,445.318,173.957,18.819,153.168
C04289=1082.703,-62.958,445.306,173.959,18.820,153.168
C04290=1082.709,-62.708,445.294,173.960,18.822,153.168
C04291=1082.715,-62.459,445.284,173.961,18.823,153.168
C04292=1082.721,-62.209,445.272,173.963,18.825,153.168
C04293=1082.727,-61.960,445.261,173.964,18.826,153.168
C04294=1082.733,-61.709,445.249,173.967,18.828,153.168
C04295=1082.739,-61.460,445.238,173.968,18.830,153.168
C04296=1082.745,-61.210,445.226,173.970,18.831,153.168
C04297=1082.751,-60.961,445.215,173.971,18.833,153.168
C04298=1082.757,-60.710,445.204,173.972,18.834,153.168
C04299=1082.763,-60.461,445.192,173.974,18.836,153.168
C04300=1082.769,-60.211,445.181,173.975,18.837,153.169
C04301=1082.775,-59.962,445.169,173.977,18.839,153.169
C04302=1082.781,-59.712,445.158,173.978,18.840,153.169
C04303=1082.787,-59.462,445.147,173.980,18.842,153.169
C04304=1082.793,-59.213,445.134,173.981,18.844,153.169
C04305=1082.799,-58.963,445.123,173.982,18.845,153.169
C04306=1082.805,-58.714,445.111,173.984,18.847,153.169
C04307=1082.811,-58.464,445.101,173.985,18.849,153.169
C04308=1082.817,-58.214,445.088,173.987,18.850,153.169
C04309=1082.823,-57.965,445.077,173.988,18.852,153.169
C04310=1082.829,-57.714,445.066,173.989,18.853,153.169
C04311=1082.835,-57.466,445.054,173.992,18.855,153.169
C04312=1082.841,-57.215,445.042,173.993,18.857,153.169
C04313=1082.847,-56.966,445.031,173.995,18.858,153.169
C04314=1082.853,-56.716,445.020,173.996,18.860,153.169
C04315=1082.859,-56.467,445.008,173.997,18.861,153.169
C04316=1082.865,-56.217,444.996,173.999,18.863,153.169
C04317=1082.871,-55.967,444.984,174.000,18.864,153.169
C04318=1082.877,-55.718,444.973,174.002,18.866,153.169
C04319=1082.883,-55.468,444.961,174.003,18.868,153.169
C04320=1082.889,-55.218,444.950,174.004,18.870,153.169
C04321=1082.896,-54.969,444.938,174.006,18.871,153.169
C04322=1082.902,-54.719,444.926,174.007,18.873,153.169
C04323=1082.907,-54.469,444.915,174.009,18.874,153.170
C04324=1082.914,-54.220,444.903,174.011,18.876,153.169
C04325=1082.920,-53.970,444.892,174.013,18.878,153.170
C04326=1082.925,-53.720,444.879,174.014,18.879,153.170
C04327=1082.932,-53.470,444.868,174.015,18.881,153.170
C04328=1082.938,-53.221,444.856,174.017,18.883,153.170
C04329=1082.945,-52.972,444.844,174.018,18.884,153.170
C04330=1082.950,-52.722,444.833,174.019,18.886,153.170
C04331=1082.956,-52.472,444.821,174.021,18.887,153.170
C04332=1082.962,-52.222,444.810,174.022,18.889,153.170
C04333=1082.968,-51.973,444.797,174.024,18.890,153.170
C04334=1082.974,-51.723,444.786,174.025,18.892,153.170
C04335=1082.981,-51.473,444.774,174.027,18.893,153.170
C04336=1082.986,-51.224,444.762,174.029,18.895,153.170
C04337=1082.993,-50.974,444.750,174.030,18.898,153.170
C04338=1082.999,-50.724,444.739,174.032,18.899,153.170
C04339=1083.004,-50.475,444.727,174.033,18.901,153.170
C04340=1083.011,-50.226,444.715,174.035,18.902,153.170
C04341=1083.016,-49.976,444.703,174.036,18.904,153.170
C04342=1083.023,-49.726,444.691,174.037,18.906,153.170
C04343=1083.029,-49.453,444.678,174.039,18.907,153.171
C04344=1083.035,-49.180,444.665,174.041,18.909,153.171
C04345=1083.042,-48.907,444.652,174.042,18.911,153.171
C04346=1083.048,-48.634,444.639,174.044,18.913,153.171
C04347=1083.054,-48.385,444.627,174.045,18.914,153.171
C04348=1083.060,-48.135,444.616,174.047,18.917,153.171
C04349=1083.065,-47.885,444.603,174.048,18.918,153.171
C04350=1083.072,-47.636,444.591,174.050,18.920,153.171
C04351=1083.078,-47.386,444.579,174.051,18.922,153.171
C04352=1083.083,-47.136,444.567,174.053,18.924,153.171
C04353=1083.090,-46.887,444.555,174.054,18.925,153.171
C04354=1083.095,-46.637,444.543,174.055,18.927,153.171
C04355=1083.102,-46.388,444.531,174.057,18.929,153.171
C04356=1083.107,-46.137,444.519,174.058,18.930,153.171
C04357=1083.112,-45.888,444.507,174.060,18.932,153.171
C04358=1083.119,-45.639,444.495,174.062,18.934,153.172
C04359=1083.125,-45.389,444.483,174.063,18.936,153.172
C04360=1083.131,-45.140,444.471,174.064,18.937,153.172
C04361=1083.137,-44.889,444.459,174.066,18.939,153.172
C04362=1083.143,-44.639,444.447,174.067,18.941,153.172
C04363=1083.149,-44.390,444.435,174.069,18.942,153.172
C04364=1083.154,-44.141,444.423,174.070,18.944,153.172
C04365=1083.161,-43.891,444.411,174.071,18.946,153.172
C04366=1083.166,-43.642,444.398,174.073,18.948,153.172
C04367=1083.172,-43.391,444.387,174.075,18.949,153.172
C04368=1083.179,-43.142,444.375,174.076,18.952,153.172
C04369=1083.184,-42.893,444.362,174.078,18.953,153.172
C04370=1083.190,-42.643,444.350,174.079,18.955,153.172
C04371=1083.197,-42.393,444.338,174.080,18.957,153.173
C04372=1083.202,-42.143,444.325,174.082,18.958,153.173
C04373=1083.208,-41.894,444.313,174.083,18.960,153.173
C04374=1083.214,-41.645,444.301,174.085,18.962,153.173
C04375=1083.220,-41.394,444.289,174.087,18.964,153.173
C04376=1083.225,-41.145,444.277,174.088,18.965,153.173
C04377=1083.232,-40.895,444.265,174.089,18.967,153.173
C04378=1083.238,-40.645,444.253,174.091,18.969,153.173
C04379=1083.244,-40.395,444.240,174.092,18.970,153.173
C04380=1083.250,-40.147,444.229,174.094,18.972,153.173
C04381=1083.256,-39.897,444.216,174.096,18.974,153.173
C04382=1083.262,-39.647,444.203,174.097,18.976,153.173
C04383=1083.268,-39.397,444.191,174.098,18.978,153.173
C04384=1083.274,-39.148,444.179,174.100,18.980,153.174
C04385=1083.279,-38.898,444.167,174.101,18.981,153.174
C04386=1083.286,-38.649,444.155,174.103,18.983,153.174
C04387=1083.292,-38.399,444.142,174.104,18.985,153.174
C04388=1083.297,-38.150,444.130,174.105,18.986,153.174
C04389=1083.303,-37.900,444.117,174.107,18.989,153.174
C04390=1083.309,-37.650,444.105,174.109,18.990,153.174
C04391=1083.314,-37.401,444.093,174.110,18.992,153.174
C04392=1083.321,-37.151,444.081,174.111,18.994,153.174
C04393=1083.327,-36.901,444.068,174.113,18.995,153.174
C04394=1083.333,-36.651,444.056,174.114,18.997,153.174
C04395=1083.338,-36.402,444.043,174.115,18.999,153.174
C04396=1083.344,-36.152,444.031,174.117,19.001,153.175
C04397=1083.350,-35.902,444.018,174.119,19.003,153.175
C04398=1083.356,-35.652,444.006,174.120,19.005,153.175
C04399=1083.361,-35.403,443.994,174.122,19.007,153.175
C04400=1083.368,-35.154,443.981,174.123,19.008,153.175
C04401=1083.374,-34.904,443.968,174.124,19.010,153.175
C04402=1083.380,-34.655,443.956,174.127,19.012,153.175
C04403=1083.385,-34.405,443.944,174.128,19.014,153.175
C04404=1083.391,-34.155,443.931,174.129,19.016,153.175
C04405=1083.397,-33.906,443.919,174.130,19.018,153.175
C04406=1083.403,-33.656,443.906,174.132,19.019,153.175
C04407=1083.410,-33.383,443.892,174.134,19.022,153.176
C04408=1083.416,-33.111,443.878,174.135,19.023,153.176
C04409=1083.422,-32.838,443.866,174.137,19.025,153.176
C04410=1083.428,-32.566,443.851,174.139,19.027,153.176
C04411=1083.434,-32.316,443.839,174.140,19.029,153.176
C04412=1083.441,-32.066,443.827,174.141,19.031,153.176
C04413=1083.447,-31.817,443.814,174.143,19.033,153.176
C04414=1083.453,-31.567,443.801,174.144,19.035,153.176
C04415=1083.458,-31.318,443.789,174.145,19.037,153.176
C04416=1083.464,-31.068,443.776,174.148,19.039,153.176
C04417=1083.470,-30.818,443.764,174.149,19.040,153.176
C04418=1083.476,-30.569,443.750,174.150,19.042,153.177
C04419=1083.482,-30.319,443.738,174.152,19.044,153.177
C04420=1083.488,-30.069,443.725,174.153,19.046,153.177
C04421=1083.494,-29.820,443.713,174.154,19.047,153.177
C04422=1083.500,-29.571,443.700,174.156,19.050,153.177
C04423=1083.506,-29.321,443.687,174.158,19.051,153.177
C04424=1083.512,-29.071,443.675,174.159,19.053,153.177
C04425=1083.517,-28.821,443.662,174.160,19.055,153.177
C04426=1083.524,-28.572,443.649,174.162,19.056,153.177
C04427=1083.530,-28.322,443.636,174.163,19.058,153.177
C04428=1083.535,-28.072,443.624,174.165,19.060,153.177
C04429=1083.542,-27.823,443.612,174.167,19.063,153.178
C04430=1083.548,-27.574,443.599,174.168,19.064,153.178
C04431=1083.554,-27.324,443.586,174.169,19.066,153.178
C04432=1083.560,-27.074,443.574,174.171,19.068,153.178
C04433=1083.566,-26.825,443.561,174.172,19.070,153.178
C04434=1083.571,-26.575,443.547,174.174,19.072,153.178
C04435=1083.577,-26.325,443.535,174.175,19.074,153.178
C04436=1083.583,-26.076,443.522,174.177,19.075,153.178
C04437=1083.588,-25.826,443.509,174.178,19.077,153.178
C04438=1083.594,-25.576,443.497,174.180,19.079,153.178
C04439=1083.600,-25.327,443.484,174.182,19.081,153.179
C04440=1083.606,-25.077,443.471,174.183,19.083,153.179
C04441=1083.612,-24.828,443.457,174.184,19.085,153.179
C04442=1083.618,-24.578,443.445,174.185,19.087,153.179
C04443=1083.624,-24.328,443.432,174.187,19.088,153.179
C04444=1083.629,-24.079,443.419,174.189,19.091,153.179
C04445=1083.635,-23.830,443.407,174.190,19.093,153.179
C04446=1083.641,-23.580,443.393,174.192,19.095,153.179
C04447=1083.647,-23.330,443.380,174.193,19.096,153.179
C04448=1083.653,-23.080,443.368,174.194,19.098,153.180
C04449=1083.659,-22.831,443.354,174.196,19.100,153.180
C04450=1083.665,-22.581,443.342,174.198,19.102,153.180
C04451=1083.671,-22.332,443.329,174.199,19.104,153.180
C04452=1083.677,-22.082,443.316,174.200,19.106,153.180
C04453=1083.682,-21.832,443.302,174.202,19.108,153.180
C04454=1083.688,-21.582,443.290,174.203,19.109,153.180
C04455=1083.694,-21.334,443.277,174.205,19.112,153.180
C04456=1083.700,-21.084,443.264,174.207,19.113,153.180
C04457=1083.706,-20.835,443.251,174.208,19.115,153.181
C04458=1083.711,-20.585,443.238,174.209,19.117,153.181
C04459=1083.717,-20.335,443.224,174.210,19.119,153.181
C04460=1083.723,-20.085,443.212,174.212,19.121,153.181
C04461=1083.729,-19.836,443.199,174.214,19.123,153.181
C04462=1083.735,-19.586,443.186,174.215,19.125,153.181
C04463=1083.741,-19.337,443.172,174.217,19.127,153.181
C04464=1083.747,-19.087,443.160,174.218,19.129,153.181
C04465=1083.753,-18.838,443.146,174.220,19.131,153.181
C04466=1083.759,-18.588,443.134,174.221,19.133,153.181
C04467=1083.764,-18.338,443.120,174.223,19.134,153.182
C04468=1083.770,-18.089,443.107,174.224,19.136,153.182
C04469=1083.776,-17.839,443.094,174.225,19.138,153.182
C04470=1083.783,-17.590,443.081,174.227,19.140,153.182
C04471=1083.789,-17.316,443.066,174.229,19.142,153.182
C04472=1083.795,-17.042,443.052,174.230,19.144,153.182
C04473=1083.801,-16.769,443.037,174.232,19.146,153.182
C04474=1083.808,-16.496,443.023,174.233,19.148,153.182
C04475=1083.814,-16.246,443.010,174.235,19.150,153.183
C04476=1083.820,-15.997,442.997,174.237,19.152,153.183
C04477=1083.826,-15.747,442.983,174.238,19.155,153.183
C04478=1083.832,-15.497,442.971,174.240,19.156,153.183
C04479=1083.838,-15.248,442.957,174.241,19.158,153.183
C04480=1083.844,-14.999,442.944,174.243,19.160,153.183
C04481=1083.849,-14.749,442.931,174.244,19.162,153.183
C04482=1083.855,-14.499,442.918,174.245,19.164,153.183
C04483=1083.861,-14.250,442.904,174.247,19.166,153.183
C04484=1083.867,-14.000,442.891,174.248,19.168,153.184
C04485=1083.872,-13.750,442.877,174.250,19.170,153.184
C04486=1083.878,-13.501,442.864,174.252,19.172,153.184
C04487=1083.884,-13.251,442.852,174.253,19.174,153.184
C04488=1083.890,-13.002,442.838,174.254,19.175,153.184
C04489=1083.896,-12.752,442.824,174.256,19.178,153.184
C04490=1083.902,-12.503,442.811,174.258,19.180,153.184
C04491=1083.907,-12.253,442.798,174.259,19.181,153.184
C04492=1083.913,-12.003,442.784,174.260,19.183,153.184
C04493=1083.919,-11.754,442.771,174.261,19.185,153.185
C04494=1083.925,-11.504,442.757,174.264,19.188,153.185
C04495=1083.931,-11.254,442.743,174.265,19.190,153.185
C04496=1083.937,-11.005,442.731,174.266,19.192,153.185
C04497=1083.943,-10.755,442.717,174.268,19.193,153.185
C04498=1083.949,-10.506,442.704,174.270,19.196,153.185
C04499=1083.955,-10.256,442.690,174.271,19.197,153.185
C04500=1083.961,-10.007,442.677,174.272,19.199,153.185
C04501=1083.966,-9.757,442.663,174.274,19.201,153.186
C04502=1083.972,-9.507,442.650,174.275,19.203,153.186
C04503=1083.978,-9.258,442.636,174.277,19.205,153.186
C04504=1083.984,-9.009,442.623,174.278,19.207,153.186
C04505=1083.989,-8.759,442.609,174.280,19.209,153.186
C04506=1083.995,-8.510,442.596,174.281,19.211,153.186
C04507=1084.001,-8.260,442.583,174.283,19.213,153.186
C04508=1084.007,-8.010,442.569,174.284,19.215,153.186
C04509=1084.013,-7.760,442.555,174.286,19.217,153.186
C04510=1084.019,-7.511,442.542,174.287,19.218,153.187
C04511=1084.025,-7.261,442.528,174.289,19.221,153.187
C04512=1084.031,-7.012,442.515,174.290,19.223,153.187
C04513=1084.036,-6.762,442.501,174.292,19.225,153.187
C04514=1084.043,-6.513,442.488,174.293,19.227,153.187
C04515=1084.048,-6.264,442.474,174.294,19.229,153.187
C04516=1084.054,-6.014,442.461,174.297,19.231,153.187
C04517=1084.060,-5.764,442.446,174.298,19.233,153.187
C04518=1084.065,-5.514,442.433,174.299,19.234,153.187
C04519=1084.072,-5.265,442.420,174.300,19.236,153.188
C04520=1084.077,-5.015,442.406,174.302,19.239,153.188
C04521=1084.083,-4.766,442.393,174.304,19.240,153.188
C04522=1084.089,-4.516,442.379,174.305,19.242,153.188
C04523=1084.096,-4.266,442.365,174.307,19.244,153.188
C04524=1084.101,-4.017,442.351,174.309,19.246,153.188
C04525=1084.107,-3.767,442.338,174.310,19.248,153.188
C04526=1084.113,-3.518,442.324,174.311,19.250,153.188
C04527=1084.118,-3.268,442.310,174.313,19.252,153.189
C04528=1084.125,-3.019,442.297,174.315,19.254,153.189
C04529=1084.130,-2.769,442.283,174.316,19.256,153.189
C04530=1084.136,-2.519,442.269,174.317,19.258,153.189
C04531=1084.142,-2.269,442.255,174.318,19.260,153.189
C04532=1084.148,-2.021,442.241,174.321,19.263,153.189
C04533=1084.154,-1.771,442.227,174.322,19.264,153.189
C04534=1084.159,-1.522,442.213,174.323,19.266,153.189
C04535=1084.165,-1.247,442.199,174.325,19.269,153.190
C04536=1084.172,-0.972,442.184,174.327,19.271,153.190
C04537=1084.178,-0.696,442.168,174.329,19.273,153.190
C04538=1084.185,-0.421,442.152,174.330,19.275,153.190
C04539=1084.190,-0.172,442.138,174.331,19.277,153.190
C04540=1084.195,0.078,442.125,174.333,19.279,153.190
C04541=1084.202,0.327,442.111,174.335,19.281,153.190
C04542=1084.207,0.577,442.097,174.336,19.283,153.191
C04543=1084.213,0.827,442.083,174.337,19.285,153.191
C04544=1084.219,1.077,442.069,174.339,19.287,153.191
C04545=1084.225,1.326,442.055,174.340,19.289,153.191
C04546=1084.231,1.575,442.042,174.342,19.291,153.191
C04547=1084.236,1.825,442.028,174.343,19.293,153.191
C04548=1084.242,2.075,442.013,174.345,19.295,153.191
C04549=1084.248,2.324,442.000,174.346,19.298,153.192
C04550=1084.253,2.574,441.986,174.348,19.299,153.192
C04551=1084.259,2.823,441.971,174.350,19.302,153.192
C04552=1084.265,3.072,441.958,174.351,19.304,153.192
C04553=1084.271,3.322,441.944,174.353,19.305,153.192
C04554=1084.277,3.572,441.930,174.354,19.307,153.192
C04555=1084.283,3.821,441.915,174.356,19.310,153.192
C04556=1084.288,4.071,441.901,174.357,19.311,153.192
C04557=1084.294,4.320,441.887,174.359,19.313,153.192
C04558=1084.300,4.570,441.874,174.360,19.315,153.193
C04559=1084.306,4.819,441.859,174.362,19.318,153.193
C04560=1084.312,5.069,441.845,174.363,19.319,153.193
C04561=1084.317,5.318,441.831,174.365,19.321,153.193
C04562=1084.323,5.568,441.817,174.366,19.323,153.193
C04563=1084.329,5.817,441.803,174.368,19.325,153.193
C04564=1084.334,6.067,441.789,174.369,19.327,153.193
C04565=1084.340,6.317,441.775,174.370,19.329,153.194
C04566=1084.347,6.566,441.761,174.373,19.331,153.194
C04567=1084.352,6.815,441.747,174.374,19.333,153.194
C04568=1084.358,7.065,441.733,174.375,19.335,153.194
C04569=1084.364,7.315,441.718,174.377,19.337,153.194
C04570=1084.370,7.564,441.704,174.379,19.340,153.194
C04571=1084.375,7.814,441.690,174.380,19.342,153.194
C04572=1084.381,8.063,441.676,174.381,19.343,153.194
C04573=1084.387,8.313,441.661,174.383,19.345,153.194
C04574=1084.393,8.563,441.648,174.385,19.348,153.195
C04575=1084.399,8.811,441.634,174.386,19.349,153.195
C04576=1084.405,9.062,441.619,174.387,19.351,153.195
C04577=1084.411,9.311,441.605,174.389,19.354,153.195
C04578=1084.416,9.560,441.591,174.391,19.355,153.195
C04579=1084.423,9.810,441.577,174.392,19.357,153.195
C04580=1084.428,10.059,441.562,174.393,19.359,153.195
C04581=1084.434,10.309,441.548,174.396,19.361,153.195
C04582=1084.440,10.559,441.533,174.397,19.363,153.196
C04583=1084.446,10.808,441.519,174.398,19.365,153.196
C04584=1084.451,11.058,441.506,174.400,19.367,153.196
C04585=1084.458,11.307,441.491,174.402,19.369,153.196
C04586=1084.463,11.557,441.477,174.403,19.371,153.196
C04587=1084.469,11.807,441.462,174.404,19.373,153.196
C04588=1084.475,12.056,441.448,174.406,19.375,153.196
C04589=1084.481,12.305,441.433,174.408,19.377,153.196
C04590=1084.487,12.555,441.420,174.409,19.379,153.196
C04591=1084.493,12.804,441.405,174.411,19.381,153.197
C04592=1084.499,13.054,441.391,174.412,19.383,153.197
C04593=1084.505,13.303,441.376,174.414,19.385,153.197
C04594=1084.511,13.553,441.362,174.415,19.387,153.197
C04595=1084.517,13.803,441.347,174.417,19.390,153.197
C04596=1084.523,14.052,441.333,174.419,19.391,153.197
C04597=1084.529,14.302,441.319,174.420,19.393,153.197
C04598=1084.535,14.551,441.304,174.422,19.395,153.197
C04599=1084.540,14.828,441.288,174.423,19.397,153.198
C04600=1084.547,15.105,441.272,174.425,19.400,153.198
C04601=1084.554,15.383,441.256,174.427,19.402,153.198
C04602=1084.560,15.660,441.240,174.429,19.404,153.198
C04603=1084.565,15.909,441.225,174.430,19.406,153.198
C04604=1084.571,16.158,441.211,174.431,19.408,153.198
C04605=1084.577,16.408,441.196,174.433,19.410,153.198
C04606=1084.583,16.657,441.182,174.435,19.412,153.199
C04607=1084.589,16.907,441.167,174.436,19.414,153.199
C04608=1084.594,17.156,441.152,174.438,19.416,153.199
C04609=1084.600,17.406,441.138,174.439,19.418,153.199
C04610=1084.606,17.656,441.123,174.441,19.420,153.199
C04611=1084.612,17.905,441.109,174.443,19.422,153.199
C04612=1084.618,18.155,441.095,174.444,19.424,153.199
C04613=1084.624,18.404,441.080,174.445,19.426,153.199
C04614=1084.629,18.654,441.064,174.447,19.428,153.199
C04615=1084.635,18.903,441.050,174.449,19.430,153.200
C04616=1084.641,19.152,441.036,174.450,19.432,153.200
C04617=1084.647,19.402,441.021,174.451,19.434,153.200
C04618=1084.653,19.651,441.006,174.454,19.436,153.200
C04619=1084.658,19.902,440.992,174.455,19.438,153.200
C04620=1084.664,20.150,440.977,174.456,19.441,153.200
C04621=1084.670,20.400,440.962,174.458,19.443,153.200
C04622=1084.676,20.649,440.948,174.460,19.445,153.201
C04623=1084.681,20.899,440.933,174.461,19.447,153.201
C04624=1084.687,21.149,440.918,174.463,19.449,153.201
C04625=1084.693,21.398,440.904,174.464,19.451,153.201
C04626=1084.699,21.647,440.889,174.466,19.453,153.201
C04627=1084.704,21.897,440.874,174.468,19.455,153.201
C04628=1084.710,22.147,440.859,174.469,19.457,153.201
C04629=1084.716,22.396,440.845,174.470,19.459,153.201
C04630=1084.722,22.646,440.829,174.472,19.461,153.202
C04631=1084.728,22.895,440.815,174.474,19.463,153.202
C04632=1084.734,23.145,440.800,174.475,19.465,153.202
C04633=1084.739,23.394,440.785,174.476,19.467,153.202
C04634=1084.745,23.643,440.771,174.479,19.469,153.202
C04635=1084.751,23.893,440.756,174.480,19.471,153.202
C04636=1084.756,24.142,440.740,174.481,19.473,153.202
C04637=1084.762,24.392,440.725,174.483,19.475,153.202
C04638=1084.768,24.641,440.711,174.485,19.477,153.203
C04639=1084.774,24.891,440.696,174.486,19.479,153.203
C04640=1084.779,25.140,440.681,174.488,19.481,153.203
C04641=1084.786,25.390,440.667,174.489,19.483,153.203
C04642=1084.791,25.640,440.651,174.491,19.485,153.203
C04643=1084.797,25.889,440.636,174.493,19.487,153.203
C04644=1084.803,26.138,440.621,174.494,19.489,153.203
C04645=1084.809,26.388,440.606,174.495,19.491,153.203
C04646=1084.815,26.637,440.591,174.498,19.493,153.203
C04647=1084.821,26.886,440.577,174.499,19.495,153.204
C04648=1084.826,27.136,440.561,174.500,19.497,153.204
C04649=1084.832,27.385,440.547,174.502,19.499,153.204
C04650=1084.838,27.635,440.531,174.504,19.501,153.204
C04651=1084.844,27.884,440.517,174.505,19.503,153.204
C04652=1084.850,28.134,440.502,174.507,19.505,153.204
C04653=1084.855,28.383,440.486,174.508,19.507,153.204
C04654=1084.861,28.633,440.471,174.510,19.509,153.205
C04655=1084.867,28.883,440.456,174.512,19.511,153.205
C04656=1084.873,29.132,440.441,174.513,19.513,153.205
C04657=1084.878,29.382,440.426,174.514,19.515,153.205
C04658=1084.884,29.631,440.411,174.517,19.518,153.205
C04659=1084.890,29.881,440.396,174.518,19.519,153.205
C04660=1084.896,30.130,440.381,174.519,19.521,153.205
C04661=1084.901,30.380,440.366,174.521,19.524,153.205
C04662=1084.907,30.628,440.351,174.523,19.525,153.205
C04663=1084.913,30.908,440.334,174.525,19.528,153.206
C04664=1084.920,31.186,440.317,174.526,19.530,153.206
C04665=1084.926,31.464,440.300,174.528,19.532,153.206
C04666=1084.933,31.743,440.284,174.530,19.535,153.206
C04667=1084.938,31.993,440.268,174.532,19.536,153.206
C04668=1084.943,32.242,440.253,174.533,19.538,153.206
C04669=1084.950,32.492,440.238,174.535,19.541,153.206
C04670=1084.956,32.741,440.222,174.536,19.542,153.206
C04671=1084.961,32.990,440.207,174.538,19.544,153.207
C04672=1084.967,33.240,440.192,174.540,19.547,153.207
C04673=1084.973,33.489,440.177,174.541,19.548,153.207
C04674=1084.978,33.739,440.161,174.542,19.550,153.207
C04675=1084.984,33.989,440.146,174.545,19.553,153.207
C04676=1084.990,34.238,440.131,174.546,19.554,153.207
C04677=1084.996,34.487,440.115,174.547,19.556,153.207
C04678=1085.002,34.737,440.100,174.549,19.559,153.207
C04679=1085.007,34.986,440.085,174.551,19.560,153.208
C04680=1085.013,35.236,440.069,174.552,19.562,153.208
C04681=1085.019,35.485,440.055,174.554,19.565,153.208
C04682=1085.025,35.734,440.039,174.556,19.566,153.208
C04683=1085.031,35.984,440.024,174.558,19.569,153.208
C04684=1085.036,36.233,440.008,174.559,19.570,153.208
C04685=1085.042,36.483,439.993,174.560,19.572,153.208
C04686=1085.048,36.732,439.977,174.562,19.575,153.208
C04687=1085.053,36.981,439.962,174.564,19.576,153.208
C04688=1085.060,37.231,439.947,174.565,19.578,153.209
C04689=1085.066,37.481,439.932,174.567,19.580,153.209
C04690=1085.071,37.730,439.916,174.569,19.582,153.209
C04691=1085.077,37.979,439.901,174.570,19.584,153.209
C04692=1085.083,38.229,439.885,174.572,19.586,153.209
C04693=1085.088,38.478,439.869,174.573,19.588,153.209
C04694=1085.094,38.728,439.854,174.576,19.591,153.209
C04695=1085.100,38.978,439.839,174.577,19.593,153.209
C04696=1085.106,39.226,439.823,174.578,19.595,153.210
C04697=1085.111,39.476,439.807,174.580,19.597,153.210
C04698=1085.117,39.726,439.792,174.582,19.599,153.210
C04699=1085.122,39.975,439.776,174.583,19.601,153.210
C04700=1085.129,40.224,439.761,174.585,19.603,153.210
C04701=1085.134,40.474,439.745,174.587,19.605,153.210
C04702=1085.140,40.723,439.730,174.589,19.607,153.210
C04703=1085.145,40.973,439.714,174.590,19.609,153.210
C04704=1085.151,41.223,439.698,174.591,19.611,153.210
C04705=1085.157,41.471,439.683,174.593,19.613,153.211
C04706=1085.163,41.721,439.668,174.595,19.615,153.211
C04707=1085.169,41.971,439.651,174.596,19.617,153.211
C04708=1085.174,42.221,439.636,174.598,19.619,153.211
C04709=1085.180,42.469,439.620,174.600,19.621,153.211
C04710=1085.186,42.719,439.605,174.602,19.623,153.211
C04711=1085.192,42.969,439.589,174.603,19.625,153.211
C04712=1085.197,43.218,439.574,174.604,19.627,153.211
C04713=1085.203,43.467,439.558,174.607,19.629,153.212
C04714=1085.209,43.717,439.542,174.608,19.631,153.212
C04715=1085.214,43.967,439.526,174.610,19.633,153.212
C04716=1085.220,44.215,439.510,174.611,19.635,153.212
C04717=1085.225,44.465,439.495,174.613,19.637,153.212
C04718=1085.231,44.715,439.479,174.615,19.639,153.212
C04719=1085.236,44.964,439.463,174.616,19.641,153.212
C04720=1085.242,45.213,439.447,174.618,19.643,153.212
C04721=1085.248,45.463,439.432,174.620,19.645,153.212
C04722=1085.254,45.713,439.415,174.621,19.647,153.213
C04723=1085.259,45.962,439.400,174.623,19.649,153.213
C04724=1085.265,46.211,439.384,174.624,19.651,153.213
C04725=1085.271,46.461,439.368,174.626,19.653,153.213
C04726=1085.276,46.710,439.352,174.628,19.655,153.213
C04727=1085.282,46.989,439.334,174.630,19.658,153.213
C04728=1085.289,47.267,439.317,174.631,19.660,153.213
C04729=1085.295,47.545,439.299,174.633,19.662,153.213
C04730=1085.301,47.824,439.281,174.635,19.665,153.214
C04731=1085.307,48.073,439.266,174.637,19.666,153.214
C04732=1085.313,48.323,439.250,174.638,19.668,153.214
C04733=1085.319,48.573,439.234,174.641,19.670,153.214
C04734=1085.324,48.821,439.218,174.642,19.672,153.214
C04735=1085.330,49.071,439.202,174.644,19.675,153.214
C04736=1085.336,49.321,439.186,174.645,19.676,153.214
C04737=1085.341,49.570,439.170,174.647,19.678,153.214
C04738=1085.347,49.820,439.153,174.649,19.680,153.214
C04739=1085.352,50.069,439.138,174.650,19.682,153.215
C04740=1085.358,50.318,439.122,174.652,19.685,153.215
C04741=1085.364,50.568,439.105,174.654,19.686,153.215
C04742=1085.369,50.818,439.090,174.655,19.688,153.215
C04743=1085.375,51.067,439.074,174.657,19.690,153.215
C04744=1085.381,51.316,439.058,174.658,19.692,153.215
C04745=1085.387,51.565,439.042,174.661,19.694,153.215
C04746=1085.392,51.815,439.026,174.662,19.696,153.215
C04747=1085.398,52.064,439.010,174.663,19.698,153.216
C04748=1085.404,52.314,438.993,174.666,19.700,153.215
C04749=1085.410,52.563,438.977,174.667,19.702,153.216
C04750=1085.414,52.813,438.961,174.669,19.704,153.216
C04751=1085.420,53.062,438.945,174.670,19.706,153.216
C04752=1085.426,53.311,438.929,174.672,19.708,153.216
C04753=1085.432,53.561,438.913,174.674,19.710,153.216
C04754=1085.438,53.810,438.896,174.675,19.712,153.216
C04755=1085.444,54.060,438.881,174.677,19.714,153.216
C04756=1085.450,54.309,438.865,174.679,19.716,153.216
C04757=1085.455,54.558,438.849,174.681,19.718,153.216
C04758=1085.460,54.808,438.832,174.682,19.720,153.217
C04759=1085.466,55.057,438.816,174.684,19.722,153.217
C04760=1085.472,55.306,438.799,174.686,19.724,153.217
C04761=1085.478,55.556,438.784,174.687,19.726,153.217
C04762=1085.484,55.806,438.768,174.689,19.728,153.217
C04763=1085.490,56.055,438.751,174.691,19.730,153.217
C04764=1085.496,56.304,438.735,174.693,19.732,153.217
C04765=1085.501,56.554,438.718,174.694,19.734,153.217
C04766=1085.507,56.803,438.702,174.696,19.735,153.217
C04767=1085.513,57.053,438.686,174.698,19.738,153.217
C04768=1085.518,57.301,438.670,174.699,19.739,153.217
C04769=1085.524,57.551,438.654,174.702,19.742,153.218
C04770=1085.530,57.800,438.637,174.703,19.743,153.218
C04771=1085.535,58.050,438.621,174.704,19.745,153.218
C04772=1085.541,58.300,438.605,174.707,19.747,153.218
C04773=1085.547,58.549,438.589,174.708,19.749,153.218
C04774=1085.553,58.798,438.572,174.710,19.751,153.218
C04775=1085.559,59.048,438.556,174.711,19.753,153.218
C04776=1085.565,59.297,438.540,174.714,19.755,153.218
C04777=1085.570,59.547,438.523,174.715,19.757,153.218
C04778=1085.576,59.796,438.507,174.716,19.759,153.218
C04779=1085.582,60.045,438.491,174.719,19.761,153.218
C04780=1085.588,60.295,438.474,174.720,19.763,153.219
C04781=1085.593,60.544,438.457,174.722,19.765,153.219
C04782=1085.599,60.794,438.441,174.724,19.767,153.219
C04783=1085.605,61.043,438.425,174.726,19.769,153.219
C04784=1085.611,61.292,438.408,174.727,19.770,153.219
C04785=1085.617,61.541,438.392,174.729,19.773,153.219
C04786=1085.622,61.791,438.375,174.731,19.774,153.219
C04787=1085.628,62.040,438.359,174.732,19.776,153.219
C04788=1085.634,62.290,438.342,174.735,19.778,153.219
C04789=1085.640,62.539,438.326,174.736,19.780,153.219
C04790=1085.645,62.789,438.309,174.738,19.782,153.219
C04791=1085.652,63.067,438.290,174.740,19.784,153.219
C04792=1085.659,63.346,438.272,174.742,19.786,153.220
C04793=1085.665,63.623,438.254,174.744,19.788,153.220
C04794=1085.671,63.902,438.236,174.746,19.791,153.220
C04795=1085.677,64.151,438.219,174.748,19.792,153.220
C04796=1085.684,64.400,438.202,174.750,19.794,153.220
C04797=1085.689,64.650,438.186,174.751,19.796,153.220
C04798=1085.695,64.899,438.169,174.753,19.798,153.220
C04799=1085.701,65.148,438.153,174.755,19.800,153.220
C04800=1085.706,65.398,438.136,174.756,19.802,153.220
C04801=1085.712,65.647,438.119,174.758,19.804,153.220
C04802=1085.717,65.896,438.102,174.760,19.806,153.220
C04803=1085.723,66.146,438.086,174.762,19.808,153.220
C04804=1085.729,66.395,438.069,174.763,19.810,153.221
C04805=1085.735,66.645,438.053,174.766,19.812,153.221
C04806=1085.741,66.894,438.036,174.767,19.814,153.221
C04807=1085.747,67.144,438.019,174.769,19.816,153.221
C04808=1085.753,67.393,438.003,174.771,19.817,153.221
C04809=1085.758,67.643,437.986,174.772,19.819,153.221
C04810=1085.764,67.892,437.969,174.774,19.821,153.221
C04811=1085.769,68.141,437.952,174.775,19.823,153.221
C04812=1085.775,68.391,437.936,174.778,19.825,153.221
C04813=1085.781,68.640,437.918,174.779,19.827,153.221
C04814=1085.787,68.889,437.902,174.781,19.829,153.221
C04815=1085.792,69.139,437.885,174.783,19.831,153.221
C04816=1085.798,69.388,437.869,174.785,19.833,153.221
C04817=1085.803,69.637,437.851,174.786,19.835,153.222
C04818=1085.809,69.886,437.835,174.789,19.837,153.222
C04819=1085.815,70.136,437.818,174.790,19.838,153.222
C04820=1085.820,70.385,437.801,174.792,19.841,153.222
C04821=1085.827,70.635,437.784,174.794,19.842,153.222
C04822=1085.832,70.884,437.766,174.795,19.844,153.222
C04823=1085.838,71.134,437.750,174.797,19.846,153.222
C04824=1085.843,71.383,437.733,174.799,19.848,153.222
C04825=1085.849,71.632,437.716,174.801,19.850,153.222
C04826=1085.855,71.882,437.699,174.802,19.852,153.222
C04827=1085.860,72.131,437.682,174.805,19.854,153.222
C04828=1085.865,72.380,437.665,174.806,19.856,153.222
C04829=1085.871,72.630,437.649,174.808,19.857,153.222
C04830=1085.877,72.879,437.631,174.810,19.860,153.223
C04831=1085.884,73.129,437.615,174.812,19.861,153.223
C04832=1085.889,73.378,437.597,174.813,19.863,153.223
C04833=1085.894,73.627,437.580,174.815,19.865,153.223
C04834=1085.900,73.876,437.563,174.817,19.867,153.223
C04835=1085.906,74.126,437.546,174.819,19.869,153.223
C04836=1085.911,74.375,437.529,174.821,19.871,153.223
C04837=1085.917,74.624,437.512,174.823,19.873,153.223
C04838=1085.923,74.873,437.495,174.824,19.874,153.223
C04839=1085.929,75.124,437.478,174.826,19.877,153.223
C04840=1085.934,75.373,437.460,174.828,19.878,153.223
C04841=1085.940,75.622,437.444,174.830,19.880,153.223
C04842=1085.945,75.871,437.426,174.832,19.882,153.223
C04843=1085.951,76.121,437.409,174.834,19.884,153.224
C04844=1085.957,76.369,437.392,174.835,19.886,153.224
C04845=1085.963,76.620,437.375,174.838,19.888,153.224
C04846=1085.968,76.869,437.358,174.839,19.890,153.224
C04847=1085.975,77.118,437.341,174.841,19.892,153.224
C04848=1085.980,77.367,437.324,174.843,19.893,153.224
C04849=1085.985,77.616,437.306,174.844,19.895,153.224
C04850=1085.991,77.867,437.289,174.846,19.897,153.224
C04851=1085.997,78.115,437.272,174.848,19.899,153.224
C04852=1086.003,78.364,437.255,174.850,19.901,153.224
C04853=1086.008,78.614,437.238,174.852,19.902,153.224
C04854=1086.014,78.863,437.220,174.854,19.905,153.224
C04855=1086.020,79.141,437.201,174.856,19.907,153.224
C04856=1086.027,79.420,437.182,174.858,19.909,153.224
C04857=1086.033,79.698,437.162,174.860,19.911,153.224
C04858=1086.039,79.976,437.142,174.862,19.913,153.225
C04859=1086.045,80.226,437.126,174.864,19.915,153.225
C04860=1086.050,80.475,437.108,174.865,19.917,153.225
C04861=1086.056,80.724,437.091,174.868,19.919,153.225
C04862=1086.062,80.974,437.074,174.869,19.921,153.225
C04863=1086.067,81.223,437.056,174.871,19.923,153.225
C04864=1086.073,81.472,437.039,174.873,19.924,153.225
C04865=1086.078,81.721,437.021,174.875,19.926,153.225
C04866=1086.084,81.971,437.004,174.876,19.928,153.225
C04867=1086.090,82.221,436.986,174.879,19.930,153.225
C04868=1086.095,82.470,436.969,174.880,19.932,153.225
C04869=1086.101,82.719,436.951,174.882,19.934,153.225
C04870=1086.106,82.968,436.934,174.884,19.936,153.225
C04871=1086.113,83.218,436.917,174.886,19.938,153.225
C04872=1086.118,83.467,436.899,174.888,19.939,153.225
C04873=1086.124,83.716,436.882,174.890,19.941,153.225
C04874=1086.129,83.965,436.864,174.891,19.943,153.226
C04875=1086.135,84.215,436.847,174.894,19.945,153.226
C04876=1086.141,84.464,436.829,174.895,19.946,153.226
C04877=1086.146,84.713,436.812,174.897,19.948,153.226
C04878=1086.152,84.963,436.794,174.899,19.950,153.226
C04879=1086.158,85.212,436.776,174.901,19.952,153.226
C04880=1086.163,85.461,436.759,174.902,19.954,153.226
C04881=1086.169,85.710,436.741,174.905,19.956,153.226
C04882=1086.175,85.960,436.723,174.906,19.957,153.226
C04883=1086.180,86.210,436.706,174.909,19.959,153.226
C04884=1086.186,86.459,436.689,174.911,19.962,153.226
C04885=1086.192,86.708,436.671,174.912,19.963,153.226
C04886=1086.197,86.957,436.653,174.915,19.965,153.226
C04887=1086.203,87.206,436.636,174.916,19.967,153.226
C04888=1086.209,87.456,436.618,174.918,19.969,153.226
C04889=1086.215,87.705,436.600,174.920,19.970,153.226
C04890=1086.220,87.954,436.583,174.922,19.972,153.226
C04891=1086.226,88.204,436.565,174.924,19.974,153.226
C04892=1086.232,88.453,436.547,174.926,19.976,153.226
C04893=1086.237,88.702,436.530,174.927,19.978,153.226
C04894=1086.243,88.952,436.512,174.930,19.980,153.226
C04895=1086.249,89.201,436.494,174.931,19.981,153.227
C04896=1086.255,89.451,436.476,174.933,19.983,153.227
C04897=1086.260,89.700,436.459,174.935,19.985,153.227
C04898=1086.266,89.949,436.441,174.937,19.987,153.227
C04899=1086.272,90.198,436.423,174.940,19.989,153.227
C04900=1086.278,90.447,436.406,174.941,19.990,153.227
C04901=1086.284,90.697,436.388,174.943,19.992,153.227
C04902=1086.289,90.946,436.370,174.945,19.993,153.227
C04903=1086.294,91.196,436.352,174.947,19.996,153.227
C04904=1086.300,91.445,436.334,174.948,19.997,153.227
C04905=1086.306,91.694,436.316,174.951,19.999,153.227
C04906=1086.311,91.943,436.299,174.952,20.001,153.227
C04907=1086.318,92.192,436.280,174.955,20.003,153.227
C04908=1086.322,92.442,436.262,174.956,20.004,153.227
C04909=1086.328,92.691,436.244,174.958,20.006,153.227
C04910=1086.334,92.941,436.227,174.960,20.009,153.227
C04911=1086.340,93.190,436.209,174.962,20.010,153.227
C04912=1086.345,93.440,436.190,174.964,20.012,153.227
C04913=1086.350,93.689,436.173,174.966,20.014,153.227
C04914=1086.356,93.937,436.155,174.968,20.016,153.227
C04915=1086.362,94.187,436.137,174.970,20.017,153.227
C04916=1086.367,94.436,436.119,174.972,20.019,153.227
C04917=1086.373,94.686,436.101,174.973,20.021,153.227
C04918=1086.379,94.935,436.083,174.976,20.023,153.227
C04919=1086.385,95.213,436.063,174.978,20.025,153.227
C04920=1086.392,95.491,436.043,174.980,20.027,153.228
C04921=1086.398,95.770,436.022,174.983,20.029,153.228
C04922=1086.404,96.048,436.002,174.984,20.031,153.228
C04923=1086.410,96.297,435.984,174.986,20.033,153.228
C04924=1086.416,96.546,435.966,174.988,20.034,153.228
C04925=1086.421,96.796,435.948,174.990,20.036,153.228
C04926=1086.427,97.046,435.930,174.993,20.038,153.228
C04927=1086.433,97.294,435.912,174.994,20.039,153.228
C04928=1086.438,97.544,435.893,174.996,20.041,153.228
C04929=1086.443,97.793,435.876,174.998,20.043,153.228
C04930=1086.449,98.041,435.857,175.000,20.045,153.228
C04931=1086.455,98.291,435.839,175.002,20.046,153.228
C04932=1086.460,98.541,435.821,175.004,20.048,153.228
C04933=1086.467,98.790,435.803,175.006,20.050,153.228
C04934=1086.472,99.039,435.785,175.008,20.052,153.228
C04935=1086.478,99.289,435.766,175.010,20.054,153.228
C04936=1086.483,99.537,435.748,175.012,20.055,153.228
C04937=1086.489,99.787,435.730,175.014,20.057,153.228
C04938=1086.494,100.036,435.712,175.015,20.059,153.228
C04939=1086.501,100.285,435.693,175.018,20.061,153.228
C04940=1086.507,100.535,435.675,175.020,20.063,153.228
C04941=1086.512,100.784,435.657,175.022,20.064,153.228
C04942=1086.518,101.034,435.639,175.024,20.066,153.228
C04943=1086.524,101.283,435.621,175.025,20.068,153.228
C04944=1086.529,101.532,435.602,175.028,20.070,153.228
C04945=1086.535,101.781,435.584,175.030,20.072,153.228
C04946=1086.540,102.031,435.565,175.032,20.073,153.228
C04947=1086.545,102.280,435.547,175.034,20.075,153.228
C04948=1086.552,102.529,435.528,175.035,20.077,153.228
C04949=1086.556,102.778,435.510,175.038,20.078,153.228
C04950=1086.563,103.027,435.491,175.039,20.080,153.228
C04951=1086.568,103.277,435.473,175.042,20.082,153.228
C04952=1086.574,103.526,435.455,175.044,20.084,153.228
C04953=1086.579,103.775,435.436,175.045,20.085,153.228
C04954=1086.585,104.024,435.418,175.048,20.087,153.228
C04955=1086.590,104.274,435.400,175.049,20.088,153.228
C04956=1086.596,104.523,435.381,175.052,20.090,153.228
C04957=1086.601,104.772,435.363,175.054,20.092,153.228
C04958=1086.608,105.021,435.344,175.056,20.094,153.228
C04959=1086.613,105.270,435.325,175.058,20.096,153.228
C04960=1086.619,105.520,435.307,175.059,20.097,153.228
C04961=1086.625,105.769,435.288,175.062,20.099,153.228
C04962=1086.629,106.019,435.270,175.064,20.101,153.228
C04963=1086.636,106.268,435.251,175.066,20.103,153.228
C04964=1086.641,106.516,435.232,175.068,20.105,153.228
C04965=1086.647,106.766,435.214,175.069,20.106,153.228
C04966=1086.653,107.016,435.195,175.072,20.108,153.228
C04967=1086.657,107.265,435.177,175.074,20.110,153.228
C04968=1086.664,107.514,435.158,175.076,20.111,153.228
C04969=1086.669,107.763,435.140,175.078,20.113,153.228
C04970=1086.675,108.013,435.122,175.080,20.114,153.228
C04971=1086.681,108.262,435.102,175.082,20.116,153.228
C04972=1086.687,108.510,435.084,175.084,20.118,153.228
C04973=1086.692,108.761,435.066,175.086,20.119,153.228
C04974=1086.697,109.009,435.047,175.088,20.121,153.228
C04975=1086.703,109.258,435.028,175.091,20.123,153.228
C04976=1086.709,109.508,435.009,175.092,20.125,153.228
C04977=1086.714,109.757,434.991,175.095,20.127,153.228
C04978=1086.720,110.006,434.972,175.096,20.128,153.229
C04979=1086.726,110.256,434.953,175.099,20.130,153.228
C04980=1086.732,110.504,434.934,175.101,20.132,153.228
C04981=1086.737,110.754,434.916,175.102,20.133,153.228
C04982=1086.743,111.004,434.897,175.105,20.135,153.228
C04983=1086.750,111.281,434.876,175.107,20.137,153.228
C04984=1086.756,111.560,434.855,175.110,20.139,153.228
C04985=1086.762,111.839,434.834,175.112,20.141,153.228
C04986=1086.768,112.116,434.812,175.114,20.143,153.228
C04987=1086.774,112.366,434.794,175.116,20.144,153.228
C04988=1086.779,112.615,434.775,175.118,20.146,153.228
C04989=1086.785,112.864,434.756,175.120,20.147,153.228
C04990=1086.791,113.114,434.737,175.122,20.149,153.228
C04991=1086.797,113.362,434.719,175.125,20.151,153.228
C04992=1086.802,113.611,434.699,175.126,20.152,153.228
C04993=1086.808,113.861,434.680,175.128,20.154,153.228
C04994=1086.813,114.111,434.662,175.131,20.156,153.228
C04995=1086.819,114.359,434.643,175.133,20.157,153.228
C04996=1086.825,114.609,434.624,175.135,20.159,153.228
C04997=1086.830,114.858,434.605,175.137,20.161,153.228
C04998=1086.836,115.107,434.586,175.139,20.163,153.228
C04999=1086.841,115.356,434.567,175.141,20.165,153.228
C05000=1086.847,115.606,434.547,175.143,20.166,153.228
C05001=1086.852,115.855,434.529,175.145,20.168,153.228
C05002=1086.858,116.104,434.509,175.147,20.170,153.228
C05003=1086.863,116.353,434.490,175.149,20.171,153.228
C05004=1086.868,116.602,434.471,175.151,20.173,153.228
C05005=1086.874,116.852,434.452,175.154,20.175,153.228
C05006=1086.880,117.101,434.433,175.155,20.176,153.228
C05007=1086.885,117.350,434.414,175.158,20.178,153.228
C05008=1086.891,117.599,434.395,175.160,20.180,153.228
C05009=1086.896,117.849,434.375,175.161,20.181,153.228
C05010=1086.902,118.098,434.356,175.164,20.183,153.228
C05011=1086.907,118.347,434.337,175.166,20.185,153.228
C05012=1086.913,118.596,434.318,175.168,20.186,153.228
C05013=1086.918,118.846,434.299,175.170,20.188,153.228
C05014=1086.924,119.094,434.280,175.173,20.190,153.228
C05015=1086.929,119.344,434.261,175.174,20.191,153.228
C05016=1086.935,119.593,434.241,175.177,20.193,153.228
C05017=1086.941,119.843,434.222,175.179,20.195,153.228
C05018=1086.946,120.091,434.203,175.181,20.196,153.228
C05019=1086.952,120.340,434.183,175.183,20.198,153.228
C05020=1086.957,120.590,434.164,175.185,20.200,153.228
C05021=1086.963,120.839,434.145,175.187,20.202,153.228
C05022=1086.969,121.089,434.126,175.189,20.203,153.228
C05023=1086.974,121.337,434.107,175.192,20.205,153.228
C05024=1086.980,121.587,434.087,175.193,20.206,153.228
C05025=1086.986,121.836,434.068,175.196,20.208,153.228
C05026=1086.991,122.085,434.048,175.198,20.210,153.228
C05027=1086.997,122.334,434.029,175.200,20.211,153.228
C05028=1087.002,122.583,434.010,175.202,20.213,153.228
C05029=1087.008,122.833,433.991,175.205,20.215,153.228
C05030=1087.014,123.081,433.971,175.206,20.216,153.228
C05031=1087.019,123.331,433.952,175.209,20.218,153.228
C05032=1087.025,123.580,433.932,175.211,20.220,153.228
C05033=1087.030,123.829,433.914,175.213,20.221,153.228
C05034=1087.036,124.078,433.894,175.215,20.223,153.228
C05035=1087.042,124.327,433.874,175.217,20.225,153.228
C05036=1087.048,124.577,433.855,175.219,20.226,153.228
C05037=1087.053,124.825,433.835,175.221,20.228,153.228
C05038=1087.058,125.075,433.815,175.224,20.229,153.228
C05039=1087.064,125.325,433.796,175.226,20.230,153.228
C05040=1087.070,125.573,433.776,175.228,20.232,153.228
C05041=1087.075,125.822,433.757,175.230,20.234,153.228
C05042=1087.081,126.072,433.738,175.232,20.235,153.228
C05043=1087.087,126.320,433.718,175.235,20.237,153.228
C05044=1087.093,126.570,433.699,175.237,20.239,153.228
C05045=1087.098,126.819,433.680,175.239,20.240,153.227
C05046=1087.104,127.068,433.660,175.241,20.242,153.227
C05047=1087.110,127.347,433.637,175.243,20.244,153.227
C05048=1087.117,127.625,433.615,175.246,20.245,153.227
C05049=1087.123,127.903,433.594,175.248,20.247,153.227
C05050=1087.129,128.181,433.572,175.251,20.249,153.227
C05051=1087.135,128.430,433.553,175.253,20.251,153.227
C05052=1087.141,128.680,433.534,175.256,20.252,153.227
C05053=1087.146,128.929,433.513,175.257,20.253,153.227
C05054=1087.151,129.178,433.494,175.260,20.255,153.227
C05055=1087.157,129.427,433.474,175.262,20.257,153.227
C05056=1087.163,129.677,433.455,175.264,20.258,153.227
C05057=1087.169,129.925,433.435,175.266,20.260,153.227
C05058=1087.175,130.175,433.415,175.269,20.261,153.227
C05059=1087.181,130.424,433.395,175.271,20.263,153.227
C05060=1087.186,130.673,433.376,175.273,20.264,153.227
C05061=1087.192,130.922,433.356,175.275,20.266,153.227
C05062=1087.197,131.172,433.336,175.278,20.268,153.227
C05063=1087.203,131.420,433.316,175.279,20.269,153.227
C05064=1087.209,131.669,433.297,175.282,20.271,153.227
C05065=1087.214,131.919,433.277,175.284,20.272,153.226
C05066=1087.220,132.168,433.257,175.287,20.274,153.226
C05067=1087.226,132.417,433.237,175.288,20.275,153.226
C05068=1087.232,132.666,433.218,175.291,20.277,153.226
C05069=1087.237,132.916,433.198,175.293,20.278,153.226
C05070=1087.243,133.165,433.178,175.295,20.280,153.226
C05071=1087.248,133.414,433.157,175.297,20.281,153.226
C05072=1087.254,133.663,433.138,175.300,20.283,153.226
C05073=1087.260,133.912,433.118,175.302,20.285,153.226
C05074=1087.265,134.161,433.097,175.304,20.286,153.226
C05075=1087.271,134.410,433.078,175.306,20.288,153.226
C05076=1087.276,134.660,433.058,175.309,20.289,153.226
C05077=1087.282,134.908,433.038,175.311,20.291,153.226
C05078=1087.288,135.158,433.018,175.313,20.292,153.226
C05079=1087.293,135.407,432.998,175.315,20.294,153.226
C05080=1087.299,135.656,432.978,175.318,20.296,153.226
C05081=1087.304,135.906,432.958,175.320,20.298,153.226
C05082=1087.310,136.154,432.938,175.322,20.298,153.226
C05083=1087.316,136.403,432.918,175.324,20.300,153.226
C05084=1087.321,136.652,432.898,175.327,20.302,153.226
C05085=1087.327,136.902,432.878,175.329,20.303,153.225
C05086=1087.332,137.151,432.858,175.331,20.305,153.225
C05087=1087.338,137.400,432.838,175.334,20.306,153.225
C05088=1087.343,137.649,432.817,175.336,20.308,153.225
C05089=1087.349,137.898,432.797,175.338,20.309,153.225
C05090=1087.354,138.147,432.777,175.340,20.311,153.225
C05091=1087.360,138.396,432.758,175.343,20.313,153.225
C05092=1087.366,138.645,432.737,175.345,20.314,153.225
C05093=1087.372,138.895,432.717,175.347,20.315,153.225
C05094=1087.378,139.144,432.696,175.349,20.317,153.225
C05095=1087.383,139.393,432.677,175.352,20.319,153.225
C05096=1087.388,139.642,432.656,175.354,20.320,153.225
C05097=1087.394,139.891,432.636,175.356,20.321,153.225
C05098=1087.400,140.140,432.616,175.358,20.323,153.225
C05099=1087.406,140.389,432.596,175.361,20.325,153.225
C05100=1087.411,140.638,432.575,175.363,20.326,153.225
C05101=1087.417,140.887,432.555,175.366,20.328,153.224
C05102=1087.422,141.136,432.535,175.367,20.329,153.224
C05103=1087.427,141.385,432.514,175.370,20.331,153.224
C05104=1087.433,141.634,432.494,175.372,20.333,153.224
C05105=1087.439,141.884,432.473,175.375,20.334,153.224
C05106=1087.445,142.133,432.453,175.377,20.335,153.224
C05107=1087.450,142.383,432.434,175.379,20.337,153.224
C05108=1087.456,142.632,432.413,175.382,20.339,153.224
C05109=1087.461,142.881,432.392,175.384,20.340,153.224
C05110=1087.467,143.130,432.372,175.386,20.341,153.224
C05111=1087.473,143.408,432.349,175.389,20.343,153.224
C05112=1087.479,143.686,432.326,175.392,20.345,153.224
C05113=1087.485,143.964,432.304,175.394,20.347,153.224
C05114=1087.492,144.243,432.281,175.397,20.348,153.224
C05115=1087.498,144.492,432.260,175.399,20.350,153.223
C05116=1087.503,144.741,432.240,175.401,20.351,153.223
C05117=1087.509,144.990,432.220,175.403,20.353,153.223
C05118=1087.514,145.239,432.199,175.406,20.354,153.223
C05119=1087.520,145.487,432.178,175.408,20.356,153.223
C05120=1087.526,145.737,432.158,175.411,20.358,153.223
C05121=1087.531,145.986,432.137,175.412,20.359,153.223
C05122=1087.537,146.235,432.117,175.415,20.360,153.223
C05123=1087.542,146.484,432.096,175.417,20.362,153.223
C05124=1087.548,146.733,432.076,175.420,20.363,153.223
C05125=1087.553,146.982,432.056,175.422,20.365,153.223
C05126=1087.559,147.232,432.035,175.424,20.366,153.223
C05127=1087.565,147.480,432.014,175.427,20.367,153.222
C05128=1087.571,147.729,431.993,175.429,20.369,153.222
C05129=1087.576,147.978,431.973,175.432,20.371,153.222
C05130=1087.582,148.228,431.952,175.433,20.372,153.222
C05131=1087.587,148.477,431.931,175.436,20.373,153.222
C05132=1087.593,148.726,431.911,175.438,20.375,153.222
C05133=1087.599,148.975,431.890,175.441,20.377,153.222
C05134=1087.604,149.224,431.870,175.443,20.378,153.222
C05135=1087.610,149.474,431.849,175.446,20.380,153.222
C05136=1087.615,149.722,431.827,175.448,20.381,153.222
C05137=1087.620,149.971,431.807,175.450,20.382,153.222
C05138=1087.626,150.220,431.787,175.453,20.384,153.222
C05139=1087.632,150.470,431.766,175.455,20.385,153.221
C05140=1087.638,150.718,431.745,175.458,20.387,153.221
C05141=1087.643,150.967,431.724,175.459,20.388,153.221
C05142=1087.648,151.217,431.704,175.462,20.390,153.221
C05143=1087.655,151.466,431.682,175.464,20.391,153.221
C05144=1087.660,151.715,431.661,175.467,20.393,153.221
C05145=1087.665,151.964,431.641,175.469,20.395,153.221
C05146=1087.671,152.213,431.620,175.472,20.396,153.221
C05147=1087.676,152.462,431.599,175.474,20.397,153.221
C05148=1087.682,152.711,431.577,175.476,20.399,153.221
C05149=1087.687,152.960,431.557,175.479,20.400,153.221
C05150=1087.693,153.209,431.537,175.481,20.401,153.220
C05151=1087.699,153.458,431.515,175.484,20.403,153.221
C05152=1087.705,153.707,431.495,175.486,20.404,153.220
C05153=1087.710,153.956,431.473,175.488,20.406,153.220
C05154=1087.716,154.206,431.452,175.491,20.407,153.220
C05155=1087.721,154.455,431.432,175.493,20.409,153.220
C05156=1087.727,154.703,431.411,175.496,20.410,153.220
C05157=1087.733,154.953,431.390,175.498,20.412,153.220
C05158=1087.738,155.201,431.368,175.500,20.413,153.220
C05159=1087.744,155.451,431.348,175.502,20.415,153.220
C05160=1087.750,155.700,431.326,175.505,20.416,153.220
C05161=1087.755,155.949,431.306,175.508,20.418,153.220
C05162=1087.761,156.197,431.284,175.510,20.419,153.219
C05163=1087.766,156.447,431.264,175.513,20.420,153.219
C05164=1087.771,156.696,431.242,175.515,20.422,153.219
C05165=1087.777,156.945,431.220,175.517,20.423,153.219
C05166=1087.783,157.194,431.199,175.519,20.425,153.219
C05167=1087.788,157.443,431.178,175.522,20.426,153.219
C05168=1087.794,157.692,431.158,175.525,20.428,153.219
C05169=1087.800,157.941,431.136,175.527,20.429,153.219
C05170=1087.805,158.190,431.115,175.530,20.431,153.219
C05171=1087.811,158.439,431.094,175.532,20.432,153.218
C05172=1087.817,158.688,431.073,175.534,20.433,153.218
C05173=1087.822,158.937,431.052,175.537,20.435,153.218
C05174=1087.828,159.186,431.030,175.539,20.437,153.218
C05175=1087.833,159.465,431.007,175.542,20.438,153.218
C05176=1087.840,159.742,430.983,175.545,20.440,153.218
C05177=1087.846,160.020,430.960,175.548,20.441,153.218
C05178=1087.853,160.298,430.935,175.550,20.443,153.218
C05179=1087.858,160.547,430.914,175.553,20.444,153.218
C05180=1087.863,160.796,430.893,175.555,20.446,153.218
C05181=1087.869,161.045,430.871,175.558,20.447,153.217
C05182=1087.875,161.294,430.850,175.560,20.448,153.217
C05183=1087.881,161.543,430.829,175.562,20.450,153.217
C05184=1087.886,161.792,430.807,175.565,20.451,153.217
C05185=1087.891,162.041,430.786,175.567,20.453,153.217
C05186=1087.897,162.290,430.764,175.570,20.454,153.217
C05187=1087.902,162.539,430.743,175.572,20.456,153.217
C05188=1087.908,162.789,430.722,175.575,20.457,153.217
C05189=1087.913,163.038,430.700,175.577,20.459,153.217
C05190=1087.918,163.286,430.679,175.579,20.460,153.217
C05191=1087.924,163.535,430.657,175.582,20.461,153.216
C05192=1087.929,163.784,430.635,175.584,20.463,153.216
C05193=1087.935,164.033,430.615,175.587,20.464,153.216
C05194=1087.940,164.283,430.592,175.589,20.466,153.216
C05195=1087.946,164.531,430.571,175.592,20.468,153.216
C05196=1087.952,164.780,430.549,175.594,20.469,153.216
C05197=1087.957,165.029,430.528,175.597,20.471,153.216
C05198=1087.962,165.278,430.506,175.599,20.472,153.216
C05199=1087.968,165.527,430.484,175.602,20.474,153.216
C05200=1087.973,165.776,430.463,175.604,20.475,153.216
C05201=1087.978,166.026,430.441,175.606,20.476,153.215
C05202=1087.984,166.274,430.420,175.609,20.477,153.215
C05203=1087.989,166.524,430.398,175.611,20.479,153.215
C05204=1087.995,166.772,430.376,175.614,20.481,153.215
C05205=1088.000,167.022,430.354,175.616,20.482,153.215
C05206=1088.006,167.270,430.333,175.619,20.484,153.215
C05207=1088.011,167.519,430.311,175.622,20.485,153.215
C05208=1088.017,167.768,430.289,175.624,20.487,153.215
C05209=1088.022,168.017,430.268,175.627,20.488,153.215
C05210=1088.028,168.266,430.246,175.629,20.490,153.214
C05211=1088.033,168.515,430.225,175.632,20.491,153.214
C05212=1088.039,168.764,430.202,175.634,20.492,153.214
C05213=1088.044,169.013,430.181,175.636,20.493,153.214
C05214=1088.050,169.263,430.159,175.639,20.495,153.214
C05215=1088.055,169.511,430.138,175.641,20.496,153.214
C05216=1088.061,169.761,430.115,175.644,20.498,153.214
C05217=1088.066,170.009,430.093,175.646,20.499,153.214
C05218=1088.072,170.258,430.071,175.649,20.501,153.214
C05219=1088.077,170.507,430.049,175.652,20.502,153.213
C05220=1088.083,170.756,430.028,175.654,20.504,153.213
C05221=1088.088,171.005,430.006,175.657,20.505,153.213
C05222=1088.094,171.254,429.984,175.659,20.507,153.213
C05223=1088.099,171.503,429.962,175.662,20.508,153.213
C05224=1088.105,171.752,429.941,175.665,20.509,153.213
C05225=1088.111,172.001,429.918,175.667,20.511,153.213
C05226=1088.117,172.250,429.896,175.670,20.512,153.212
C05227=1088.122,172.499,429.874,175.672,20.513,153.212
C05228=1088.128,172.748,429.853,175.674,20.514,153.212
C05229=1088.133,172.997,429.831,175.677,20.516,153.212
C05230=1088.138,173.246,429.808,175.679,20.517,153.212
C05231=1088.145,173.495,429.786,175.682,20.519,153.212
C05232=1088.149,173.744,429.764,175.685,20.520,153.212
C05233=1088.156,173.993,429.743,175.687,20.522,153.212
C05234=1088.161,174.241,429.720,175.690,20.523,153.212
C05235=1088.166,174.491,429.698,175.692,20.524,153.211
C05236=1088.172,174.740,429.676,175.695,20.526,153.211
C05237=1088.177,174.988,429.654,175.698,20.527,153.211
C05238=1088.184,175.237,429.632,175.700,20.528,153.211
C05239=1088.189,175.515,429.608,175.703,20.530,153.211
C05240=1088.196,175.793,429.582,175.706,20.532,153.211
C05241=1088.202,176.070,429.558,175.709,20.533,153.211
C05242=1088.208,176.348,429.534,175.712,20.534,153.210
C05243=1088.214,176.597,429.511,175.714,20.536,153.210
C05244=1088.220,176.846,429.489,175.717,20.537,153.210
C05245=1088.225,177.094,429.467,175.719,20.539,153.210
C05246=1088.230,177.344,429.444,175.722,20.540,153.210
C05247=1088.237,177.593,429.423,175.725,20.541,153.210
C05248=1088.242,177.842,429.400,175.727,20.543,153.209
C05249=1088.247,178.091,429.378,175.730,20.544,153.209
C05250=1088.254,178.339,429.356,175.732,20.546,153.209
C05251=1088.259,178.589,429.333,175.735,20.547,153.209
C05252=1088.265,178.838,429.310,175.738,20.548,153.209
C05253=1088.270,179.086,429.289,175.740,20.549,153.209
C05254=1088.276,179.335,429.266,175.743,20.551,153.209
C05255=1088.281,179.584,429.244,175.746,20.552,153.209
C05256=1088.288,179.833,429.222,175.748,20.553,153.208
C05257=1088.293,180.082,429.200,175.751,20.555,153.208
C05258=1088.298,180.331,429.177,175.753,20.556,153.208
C05259=1088.305,180.580,429.155,175.756,20.558,153.208
C05260=1088.310,180.829,429.132,175.759,20.559,153.208
C05261=1088.315,181.078,429.110,175.761,20.560,153.208
C05262=1088.321,181.327,429.087,175.764,20.562,153.207
C05263=1088.327,181.576,429.066,175.767,20.563,153.207
C05264=1088.333,181.825,429.043,175.769,20.564,153.207
C05265=1088.339,182.074,429.020,175.772,20.565,153.207
C05266=1088.344,182.322,428.999,175.775,20.567,153.207
C05267=1088.350,182.571,428.976,175.777,20.568,153.207
C05268=1088.356,182.820,428.953,175.780,20.569,153.206
C05269=1088.361,183.069,428.931,175.783,20.571,153.206
C05270=1088.367,183.318,428.908,175.785,20.572,153.206
C05271=1088.373,183.567,428.885,175.788,20.573,153.206
C05272=1088.379,183.816,428.863,175.790,20.575,153.206
C05273=1088.384,184.065,428.840,175.793,20.576,153.206
C05274=1088.390,184.313,428.818,175.796,20.577,153.205
C05275=1088.396,184.563,428.796,175.798,20.579,153.205
C05276=1088.401,184.812,428.773,175.801,20.580,153.205
C05277=1088.407,185.060,428.750,175.804,20.581,153.205
C05278=1088.413,185.309,428.727,175.806,20.582,153.205
C05279=1088.418,185.558,428.705,175.809,20.584,153.205
C05280=1088.423,185.807,428.682,175.812,20.585,153.205
C05281=1088.429,186.056,428.659,175.814,20.586,153.204
C05282=1088.435,186.305,428.636,175.817,20.588,153.204
C05283=1088.440,186.554,428.614,175.819,20.589,153.204
C05284=1088.445,186.803,428.592,175.822,20.591,153.204
C05285=1088.451,187.051,428.569,175.825,20.592,153.204
C05286=1088.456,187.301,428.545,175.827,20.594,153.204
C05287=1088.462,187.550,428.522,175.830,20.595,153.204
C05288=1088.467,187.798,428.500,175.833,20.596,153.203
C05289=1088.472,188.047,428.477,175.835,20.598,153.203
C05290=1088.478,188.296,428.454,175.838,20.599,153.203
C05291=1088.484,188.545,428.431,175.841,20.601,153.203
C05292=1088.490,188.794,428.408,175.844,20.602,153.203
C05293=1088.495,189.043,428.385,175.847,20.603,153.203
C05294=1088.500,189.291,428.362,175.849,20.605,153.203
C05295=1088.505,189.540,428.339,175.852,20.606,153.202
C05296=1088.511,189.789,428.316,175.854,20.608,153.202
C05297=1088.517,190.038,428.293,175.857,20.609,153.202
C05298=1088.523,190.287,428.271,175.860,20.610,153.202
C05299=1088.528,190.536,428.247,175.862,20.612,153.202
C05300=1088.533,190.785,428.224,175.865,20.613,153.202
C05301=1088.538,191.033,428.201,175.867,20.615,153.202
C05302=1088.544,191.282,428.179,175.870,20.615,153.201
C05303=1088.551,191.560,428.153,175.874,20.617,153.201
C05304=1088.556,191.837,428.127,175.876,20.619,153.201
C05305=1088.563,192.115,428.102,175.879,20.620,153.201
C05306=1088.569,192.391,428.076,175.882,20.622,153.201
C05307=1088.575,192.640,428.053,175.885,20.623,153.201
C05308=1088.580,192.890,428.029,175.888,20.625,153.201
C05309=1088.585,193.138,428.006,175.890,20.626,153.200
C05310=1088.591,193.387,427.983,175.893,20.627,153.200
C05311=1088.597,193.636,427.961,175.896,20.629,153.200
C05312=1088.603,193.885,427.938,175.898,20.630,153.200
C05313=1088.608,194.134,427.914,175.902,20.632,153.200
C05314=1088.614,194.383,427.890,175.904,20.633,153.200
C05315=1088.619,194.632,427.867,175.907,20.634,153.199
C05316=1088.625,194.880,427.845,175.910,20.635,153.199
C05317=1088.630,195.130,427.821,175.912,20.637,153.199
C05318=1088.636,195.379,427.798,175.915,20.638,153.199
C05319=1088.642,195.627,427.775,175.918,20.639,153.199
C05320=1088.647,195.876,427.751,175.920,20.641,153.199
C05321=1088.653,196.125,427.728,175.923,20.642,153.198
C05322=1088.658,196.374,427.705,175.926,20.643,153.198
C05323=1088.664,196.623,427.682,175.928,20.645,153.198
C05324=1088.669,196.871,427.658,175.932,20.646,153.198
C05325=1088.675,197.120,427.635,175.935,20.648,153.198
C05326=1088.681,197.369,427.612,175.937,20.649,153.198
C05327=1088.686,197.618,427.588,175.940,20.650,153.197
C05328=1088.692,197.867,427.565,175.942,20.651,153.197
C05329=1088.698,198.115,427.542,175.945,20.653,153.197
C05330=1088.703,198.364,427.519,175.948,20.654,153.197
C05331=1088.709,198.613,427.494,175.950,20.655,153.197
C05332=1088.714,198.862,427.472,175.954,20.657,153.196
C05333=1088.720,199.111,427.449,175.957,20.658,153.196
C05334=1088.725,199.359,427.424,175.959,20.660,153.196
C05335=1088.731,199.608,427.401,175.962,20.661,153.196
C05336=1088.737,199.856,427.378,175.965,20.662,153.196
C05337=1088.743,200.106,427.354,175.967,20.663,153.196
C05338=1088.748,200.355,427.331,175.970,20.665,153.196
C05339=1088.755,200.604,427.307,175.973,20.666,153.195
C05340=1088.759,200.853,427.284,175.976,20.668,153.195
C05341=1088.766,201.101,427.260,175.979,20.669,153.195
C05342=1088.771,201.350,427.236,175.982,20.670,153.195
C05343=1088.777,201.599,427.213,175.984,20.671,153.195
C05344=1088.783,201.848,427.190,175.987,20.672,153.194
C05345=1088.788,202.097,427.165,175.990,20.674,153.194
C05346=1088.794,202.346,427.142,175.992,20.675,153.194
C05347=1088.800,202.594,427.119,175.996,20.677,153.194
C05348=1088.805,202.843,427.095,175.998,20.678,153.194
C05349=1088.810,203.092,427.071,176.001,20.679,153.194
C05350=1088.816,203.341,427.048,176.004,20.681,153.193
C05351=1088.821,203.589,427.024,176.006,20.682,153.193
C05352=1088.828,203.839,427.000,176.009,20.683,153.193
C05353=1088.833,204.087,426.976,176.013,20.685,153.193
C05354=1088.839,204.336,426.953,176.015,20.686,153.193
C05355=1088.844,204.585,426.929,176.018,20.687,153.193
C05356=1088.849,204.833,426.905,176.021,20.689,153.192
C05357=1088.855,205.082,426.882,176.023,20.690,153.192
C05358=1088.860,205.331,426.857,176.026,20.691,153.192
C05359=1088.866,205.580,426.833,176.029,20.693,153.192
C05360=1088.872,205.829,426.810,176.032,20.694,153.192
C05361=1088.877,206.078,426.786,176.035,20.696,153.192
C05362=1088.883,206.326,426.762,176.037,20.697,153.191
C05363=1088.888,206.575,426.738,176.040,20.698,153.191
C05364=1088.894,206.824,426.714,176.043,20.700,153.191
C05365=1088.900,207.073,426.690,176.046,20.701,153.191
C05366=1088.905,207.322,426.667,176.049,20.703,153.191
C05367=1088.928,208.345,426.568,176.120,20.739,153.187
C05368=1088.937,208.727,426.531,176.124,20.742,153.187
C05369=1088.946,209.110,426.493,176.129,20.745,153.187
C05370=1088.954,209.493,426.455,176.133,20.749,153.187
C05371=1088.963,209.875,426.418,176.137,20.752,153.187
C05372=1088.969,210.123,426.394,176.140,20.755,153.187
C05373=1088.975,210.373,426.369,176.142,20.757,153.187
C05374=1088.980,210.621,426.345,176.145,20.759,153.187
C05375=1088.985,210.870,426.320,176.148,20.762,153.187
C05376=1088.991,211.119,426.296,176.150,20.764,153.187
C05377=1088.996,211.368,426.272,176.153,20.766,153.187
C05378=1089.002,211.616,426.247,176.156,20.768,153.187
C05379=1089.008,211.865,426.222,176.159,20.770,153.187
C05380=1089.013,212.114,426.198,176.161,20.773,153.188
C05381=1089.019,212.363,426.173,176.164,20.775,153.188
C05382=1089.024,212.611,426.149,176.167,20.777,153.188
C05383=1089.031,212.860,426.123,176.170,20.780,153.188
C05384=1089.036,213.109,426.099,176.172,20.782,153.188
C05385=1089.041,213.357,426.075,176.175,20.784,153.188
C05386=1089.047,213.607,426.050,176.177,20.786,153.188
C05387=1089.053,213.855,426.025,176.181,20.789,153.188
C05388=1089.059,214.104,426.001,176.183,20.791,153.188
C05389=1089.064,214.352,425.977,176.186,20.793,153.188
C05390=1089.070,214.601,425.951,176.188,20.796,153.188
C05391=1089.075,214.850,425.926,176.191,20.798,153.188
C05392=1089.080,215.099,425.902,176.194,20.800,153.188
C05393=1089.086,215.347,425.877,176.196,20.802,153.188
C05394=1089.091,215.596,425.852,176.199,20.805,153.188
C05395=1089.097,215.845,425.828,176.202,20.807,153.188
C05396=1089.103,216.093,425.803,176.205,20.809,153.188
C05397=1089.109,216.342,425.778,176.207,20.811,153.188
C05398=1089.114,216.591,425.753,176.211,20.814,153.188
C05399=1089.120,216.840,425.728,176.213,20.816,153.189
C05400=1089.125,217.088,425.703,176.216,20.819,153.189
C05401=1089.131,217.337,425.678,176.218,20.821,153.189
C05402=1089.137,217.585,425.653,176.222,20.823,153.189
C05403=1089.143,217.834,425.629,176.224,20.825,153.189
C05404=1089.147,218.083,425.604,176.227,20.828,153.189
C05405=1089.153,218.332,425.579,176.229,20.830,153.189
C05406=1089.159,218.580,425.554,176.232,20.832,153.189
C05407=1089.165,218.829,425.529,176.235,20.834,153.189
C05408=1089.170,219.077,425.504,176.238,20.837,153.189
C05409=1089.176,219.327,425.479,176.240,20.839,153.189
C05410=1089.182,219.575,425.454,176.243,20.841,153.189
C05411=1089.187,219.824,425.429,176.246,20.843,153.189
C05412=1089.193,220.073,425.404,176.249,20.846,153.189
C05413=1089.198,220.321,425.378,176.251,20.848,153.189
C05414=1089.204,220.570,425.354,176.254,20.851,153.189
C05415=1089.210,220.818,425.329,176.257,20.853,153.189
C05416=1089.216,221.068,425.304,176.260,20.855,153.189
C05417=1089.221,221.317,425.278,176.262,20.857,153.189
C05418=1089.227,221.565,425.253,176.266,20.859,153.189
C05419=1089.233,221.814,425.229,176.268,20.861,153.189
C05420=1089.241,222.199,425.189,176.273,20.865,153.189
C05421=1089.250,222.586,425.150,176.277,20.869,153.190
C05422=1089.259,222.973,425.111,176.281,20.873,153.190
C05423=1089.267,223.359,425.071,176.285,20.876,153.190
C05424=1089.273,223.608,425.046,176.288,20.879,153.190
C05425=1089.278,223.856,425.021,176.291,20.881,153.190
C05426=1089.284,224.105,424.996,176.294,20.883,153.190
C05427=1089.290,224.354,424.970,176.296,20.885,153.190
C05428=1089.295,224.602,424.945,176.299,20.888,153.190
C05429=1089.301,224.851,424.920,176.302,20.890,153.190
C05430=1089.306,225.100,424.894,176.305,20.893,153.190
C05431=1089.312,225.348,424.869,176.308,20.895,153.190
C05432=1089.318,225.597,424.843,176.310,20.897,153.190
C05433=1089.323,225.845,424.818,176.313,20.900,153.190
C05434=1089.329,226.094,424.792,176.316,20.902,153.190
C05435=1089.335,226.343,424.767,176.319,20.904,153.190
C05436=1089.340,226.592,424.741,176.321,20.906,153.190
C05437=1089.346,226.840,424.717,176.324,20.909,153.191
C05438=1089.351,227.089,424.691,176.327,20.911,153.191
C05439=1089.357,227.338,424.665,176.330,20.913,153.191
C05440=1089.362,227.586,424.640,176.333,20.916,153.191
C05441=1089.368,227.835,424.615,176.335,20.918,153.191
C05442=1089.374,228.084,424.589,176.339,20.921,153.191
C05443=1089.379,228.333,424.563,176.341,20.923,153.191
C05444=1089.385,228.581,424.538,176.344,20.925,153.191
C05445=1089.390,228.830,424.512,176.347,20.927,153.191
C05446=1089.397,229.078,424.486,176.350,20.930,153.191
C05447=1089.402,229.327,424.460,176.352,20.932,153.191
C05448=1089.408,229.575,424.435,176.355,20.934,153.191
C05449=1089.413,229.824,424.409,176.358,20.937,153.191
C05450=1089.420,230.072,424.384,176.361,20.939,153.191
C05451=1089.425,230.321,424.358,176.364,20.942,153.191
C05452=1089.431,230.570,424.332,176.366,20.944,153.191
C05453=1089.436,230.818,424.307,176.369,20.946,153.191
C05454=1089.442,231.067,424.281,176.372,20.948,153.191
C05455=1089.447,231.316,424.255,176.375,20.951,153.191
C05456=1089.454,231.564,424.229,176.378,20.953,153.192
C05457=1089.458,231.813,424.203,176.380,20.955,153.192
C05458=1089.464,232.062,424.177,176.383,20.958,153.192
C05459=1089.469,232.311,424.151,176.386,20.960,153.192
C05460=1089.476,232.559,424.126,176.389,20.962,153.192
C05461=1089.481,232.808,424.099,176.392,20.965,153.192
C05462=1089.486,233.056,424.074,176.394,20.967,153.192
C05463=1089.492,233.305,424.048,176.398,20.970,153.192
